// NETWORK 14 (disabled)
//   axisdata[6].Axis_Inbb: A-0-0021.13 -RD- Axis is ready for power to the amplifier (bb)
//   FP_S_0_0095: Diagnostic message
//   drive6: Real axis "Drive6" with axis number 6
// fb_blink_diagnos_6(ENABLE := axisdata[6].Axis_Inbb, TIMELOW := t#1s, TIMEHIGH := t#1s); // BLINK
// fb_diagnose_6(
//     Execute := fb_blink_diagnos_6.OUT,
//     ParameterNumber := FP_S_0_0095,
//     Axis := drive6,
//     Value => str_diagnose_6); // MB_ReadStringParameter

// NETWORK 15
//   axisdata[1].Axis_Inbb: A-0-0021.13 -RD- Axis is ready for power to the amplifier (bb)
//   FP_S_0_0051: Position feedback value 1
//   drive1: Real axis "Drive1" with axis number 1
FB_readmotorencoder1(
    Enable := axisdata[1].Axis_Inbb,
    ParameterNumber := FP_S_0_0051,
    Axis := drive1,
    Value => r_motorencoder_1); // MB_ReadRealParameter

// NETWORK 16
//   axisdata[2].Axis_Inbb: A-0-0021.13 -RD- Axis is ready for power to the amplifier (bb)
//   FP_S_0_0051: Position feedback value 1
//   drive2: Real axis "Drive2" with axis number 2
FB_readmotorencoder2(
    Enable := axisdata[2].Axis_Inbb,
    ParameterNumber := FP_S_0_0051,
    Axis := drive2,
    Value => r_motorencoder_2); // MB_ReadRealParameter

// NETWORK 17
//   axisdata[3].Axis_Inbb: A-0-0021.13 -RD- Axis is ready for power to the amplifier (bb)
//   FP_S_0_0051: Position feedback value 1
//   drive3: Real axis "Drive3" with axis number 3
FB_readmotorencoder3(
    Enable := axisdata[3].Axis_Inbb,
    ParameterNumber := FP_S_0_0051,
    Axis := drive3,
    Value => r_motorencoder_3); // MB_ReadRealParameter

// NETWORK 18 (disabled)
//   axisdata[4].Axis_Inbb: A-0-0021.13 -RD- Axis is ready for power to the amplifier (bb)
//   FP_S_0_0051: Position feedback value 1
//   drive4: Real axis "Drive4" with axis number 4
// FB_readmotorencoder4(
//     Enable := axisdata[4].Axis_Inbb,
//     ParameterNumber := FP_S_0_0051,
//     Axis := drive4,
//     Value => r_motorencoder_4); // MB_ReadRealParameter

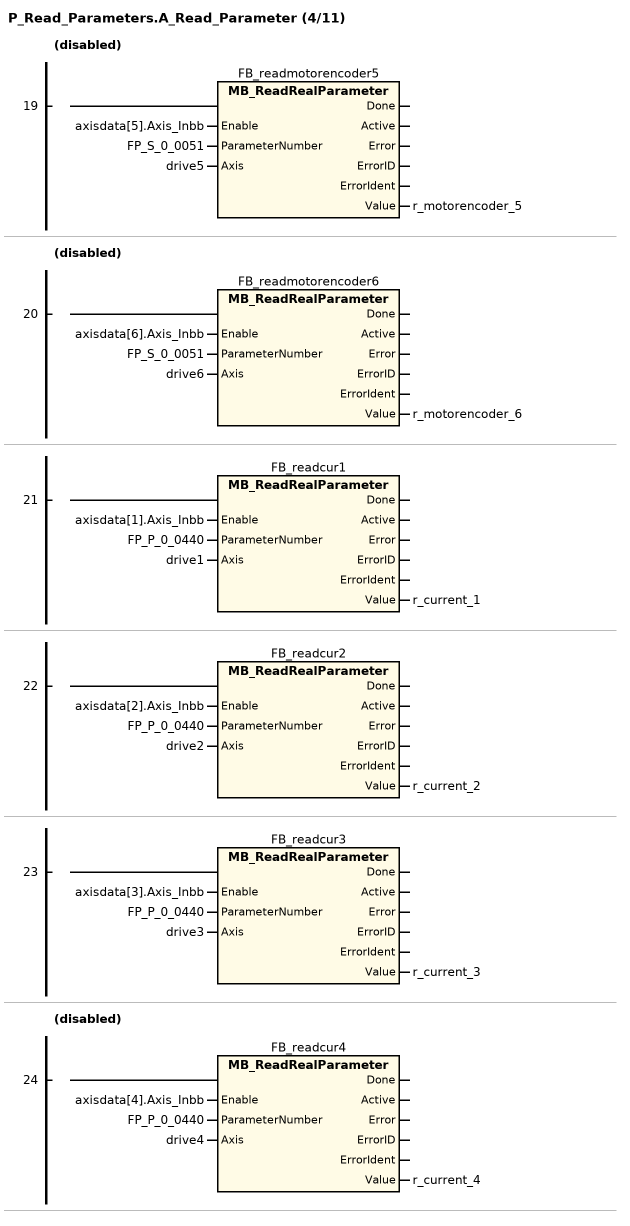
// NETWORK 19 (disabled)
//   axisdata[5].Axis_Inbb: A-0-0021.13 -RD- Axis is ready for power to the amplifier (bb)
//   FP_S_0_0051: Position feedback value 1
//   drive5: Real axis "Drive5" with axis number 5
// FB_readmotorencoder5(
//     Enable := axisdata[5].Axis_Inbb,
//     ParameterNumber := FP_S_0_0051,
//     Axis := drive5,
//     Value => r_motorencoder_5); // MB_ReadRealParameter

// NETWORK 20 (disabled)
//   axisdata[6].Axis_Inbb: A-0-0021.13 -RD- Axis is ready for power to the amplifier (bb)
//   FP_S_0_0051: Position feedback value 1
//   drive6: Real axis "Drive6" with axis number 6
// FB_readmotorencoder6(
//     Enable := axisdata[6].Axis_Inbb,
//     ParameterNumber := FP_S_0_0051,
//     Axis := drive6,
//     Value => r_motorencoder_6); // MB_ReadRealParameter

// NETWORK 21
//   FB_readcur1: With the function block "MB_ReadRealParameter" it is possible to read the current value of a parameter. The return value is REAL.
//   axisdata[1].Axis_Inbb: A-0-0021.13 -RD- Axis is ready for power to the amplifier (bb)
//   FP_P_0_0440: Actual output current value (absolute value)
//   drive1: Real axis "Drive1" with axis number 1
//   r_current_1: FP_P_0_0440,Actual output current value absolute value
FB_readcur1(
    Enable := axisdata[1].Axis_Inbb,
    ParameterNumber := FP_P_0_0440,
    Axis := drive1,
    Value => r_current_1); // MB_ReadRealParameter

// NETWORK 22
//   axisdata[2].Axis_Inbb: A-0-0021.13 -RD- Axis is ready for power to the amplifier (bb)
//   FP_P_0_0440: Actual output current value (absolute value)
//   drive2: Real axis "Drive2" with axis number 2
FB_readcur2(
    Enable := axisdata[2].Axis_Inbb,
    ParameterNumber := FP_P_0_0440,
    Axis := drive2,
    Value => r_current_2); // MB_ReadRealParameter

// NETWORK 23
//   axisdata[3].Axis_Inbb: A-0-0021.13 -RD- Axis is ready for power to the amplifier (bb)
//   FP_P_0_0440: Actual output current value (absolute value)
//   drive3: Real axis "Drive3" with axis number 3
FB_readcur3(
    Enable := axisdata[3].Axis_Inbb,
    ParameterNumber := FP_P_0_0440,
    Axis := drive3,
    Value => r_current_3); // MB_ReadRealParameter

// NETWORK 24 (disabled)
//   axisdata[4].Axis_Inbb: A-0-0021.13 -RD- Axis is ready for power to the amplifier (bb)
//   FP_P_0_0440: Actual output current value (absolute value)
//   drive4: Real axis "Drive4" with axis number 4
// FB_readcur4(
//     Enable := axisdata[4].Axis_Inbb,
//     ParameterNumber := FP_P_0_0440,
//     Axis := drive4,
//     Value => r_current_4); // MB_ReadRealParameter

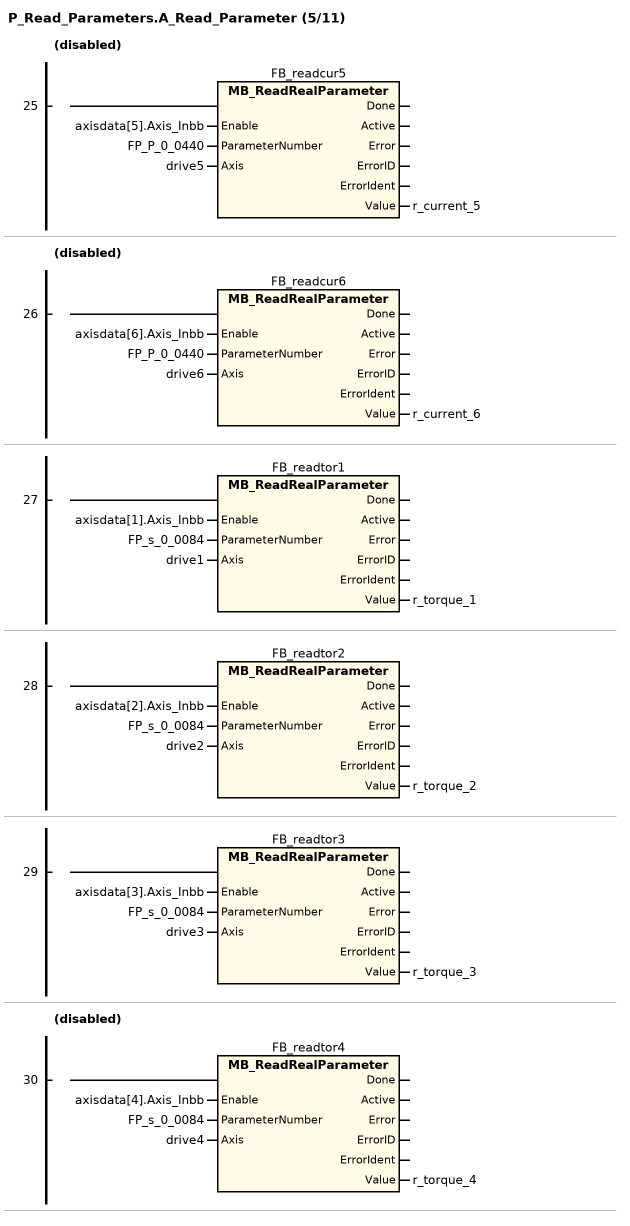
// NETWORK 25 (disabled)
//   axisdata[5].Axis_Inbb: A-0-0021.13 -RD- Axis is ready for power to the amplifier (bb)
//   FP_P_0_0440: Actual output current value (absolute value)
//   drive5: Real axis "Drive5" with axis number 5
// FB_readcur5(
//     Enable := axisdata[5].Axis_Inbb,
//     ParameterNumber := FP_P_0_0440,
//     Axis := drive5,
//     Value => r_current_5); // MB_ReadRealParameter

// NETWORK 26 (disabled)
//   axisdata[6].Axis_Inbb: A-0-0021.13 -RD- Axis is ready for power to the amplifier (bb)
//   FP_P_0_0440: Actual output current value (absolute value)
//   drive6: Real axis "Drive6" with axis number 6
// FB_readcur6(
//     Enable := axisdata[6].Axis_Inbb,
//     ParameterNumber := FP_P_0_0440,
//     Axis := drive6,
//     Value => r_current_6); // MB_ReadRealParameter

// NETWORK 27
//   axisdata[1].Axis_Inbb: A-0-0021.13 -RD- Axis is ready for power to the amplifier (bb)
//   FP_s_0_0084: Torque/force feedback value
//   drive1: Real axis "Drive1" with axis number 1
//   r_torque_1: FP_S_0_0084,Torque force feedback value
FB_readtor1(
    Enable := axisdata[1].Axis_Inbb,
    ParameterNumber := FP_s_0_0084,
    Axis := drive1,
    Value => r_torque_1); // MB_ReadRealParameter

// NETWORK 28
//   axisdata[2].Axis_Inbb: A-0-0021.13 -RD- Axis is ready for power to the amplifier (bb)
//   FP_s_0_0084: Torque/force feedback value
//   drive2: Real axis "Drive2" with axis number 2
FB_readtor2(
    Enable := axisdata[2].Axis_Inbb,
    ParameterNumber := FP_s_0_0084,
    Axis := drive2,
    Value => r_torque_2); // MB_ReadRealParameter

// NETWORK 29
//   axisdata[3].Axis_Inbb: A-0-0021.13 -RD- Axis is ready for power to the amplifier (bb)
//   FP_s_0_0084: Torque/force feedback value
//   drive3: Real axis "Drive3" with axis number 3
FB_readtor3(
    Enable := axisdata[3].Axis_Inbb,
    ParameterNumber := FP_s_0_0084,
    Axis := drive3,
    Value => r_torque_3); // MB_ReadRealParameter

// NETWORK 30 (disabled)
//   axisdata[4].Axis_Inbb: A-0-0021.13 -RD- Axis is ready for power to the amplifier (bb)
//   FP_s_0_0084: Torque/force feedback value
//   drive4: Real axis "Drive4" with axis number 4
// FB_readtor4(
//     Enable := axisdata[4].Axis_Inbb,
//     ParameterNumber := FP_s_0_0084,
//     Axis := drive4,
//     Value => r_torque_4); // MB_ReadRealParameter

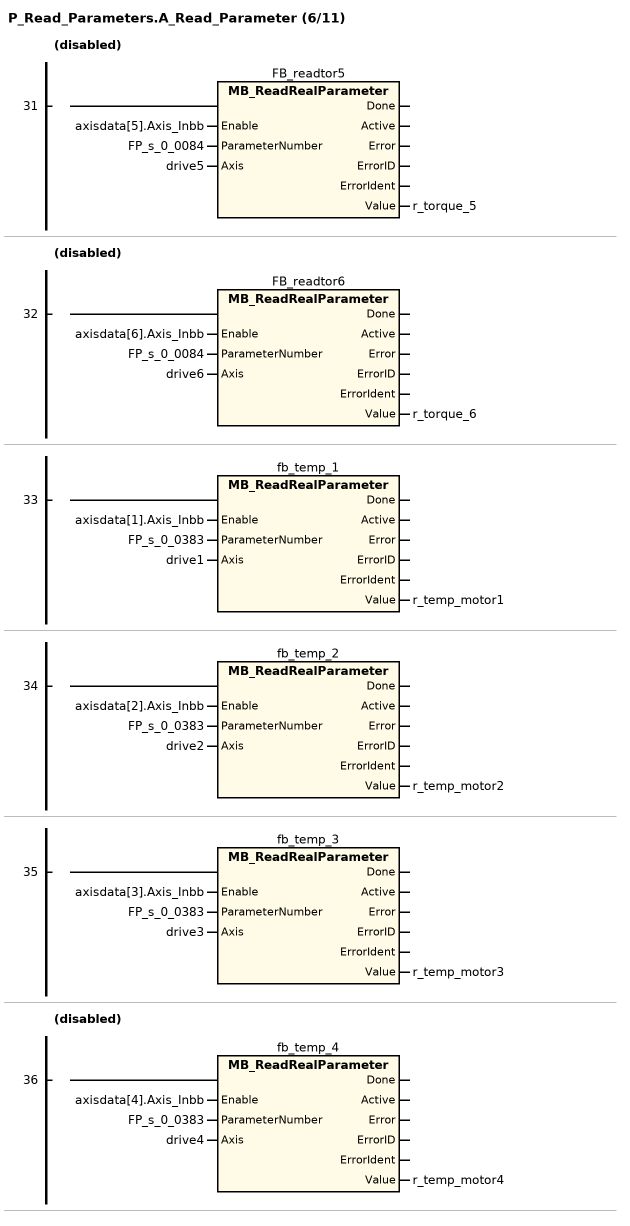
// NETWORK 31 (disabled)
//   axisdata[5].Axis_Inbb: A-0-0021.13 -RD- Axis is ready for power to the amplifier (bb)
//   FP_s_0_0084: Torque/force feedback value
//   drive5: Real axis "Drive5" with axis number 5
// FB_readtor5(
//     Enable := axisdata[5].Axis_Inbb,
//     ParameterNumber := FP_s_0_0084,
//     Axis := drive5,
//     Value => r_torque_5); // MB_ReadRealParameter

// NETWORK 32 (disabled)
//   axisdata[6].Axis_Inbb: A-0-0021.13 -RD- Axis is ready for power to the amplifier (bb)
//   FP_s_0_0084: Torque/force feedback value
//   drive6: Real axis "Drive6" with axis number 6
// FB_readtor6(
//     Enable := axisdata[6].Axis_Inbb,
//     ParameterNumber := FP_s_0_0084,
//     Axis := drive6,
//     Value => r_torque_6); // MB_ReadRealParameter

// NETWORK 33
//   axisdata[1].Axis_Inbb: A-0-0021.13 -RD- Axis is ready for power to the amplifier (bb)
//   FP_s_0_0383: Motor temperature
//   drive1: Real axis "Drive1" with axis number 1
//   r_temp_motor1: FP_S_0_0383,Motor temperature
fb_temp_1(
    Enable := axisdata[1].Axis_Inbb,
    ParameterNumber := FP_s_0_0383,
    Axis := drive1,
    Value => r_temp_motor1); // MB_ReadRealParameter

// NETWORK 34
//   axisdata[2].Axis_Inbb: A-0-0021.13 -RD- Axis is ready for power to the amplifier (bb)
//   FP_s_0_0383: Motor temperature
//   drive2: Real axis "Drive2" with axis number 2
fb_temp_2(
    Enable := axisdata[2].Axis_Inbb,
    ParameterNumber := FP_s_0_0383,
    Axis := drive2,
    Value => r_temp_motor2); // MB_ReadRealParameter

// NETWORK 35
//   axisdata[3].Axis_Inbb: A-0-0021.13 -RD- Axis is ready for power to the amplifier (bb)
//   FP_s_0_0383: Motor temperature
//   drive3: Real axis "Drive3" with axis number 3
fb_temp_3(
    Enable := axisdata[3].Axis_Inbb,
    ParameterNumber := FP_s_0_0383,
    Axis := drive3,
    Value => r_temp_motor3); // MB_ReadRealParameter

// NETWORK 36 (disabled)
//   axisdata[4].Axis_Inbb: A-0-0021.13 -RD- Axis is ready for power to the amplifier (bb)
//   FP_s_0_0383: Motor temperature
//   drive4: Real axis "Drive4" with axis number 4
// fb_temp_4(
//     Enable := axisdata[4].Axis_Inbb,
//     ParameterNumber := FP_s_0_0383,
//     Axis := drive4,
//     Value => r_temp_motor4); // MB_ReadRealParameter

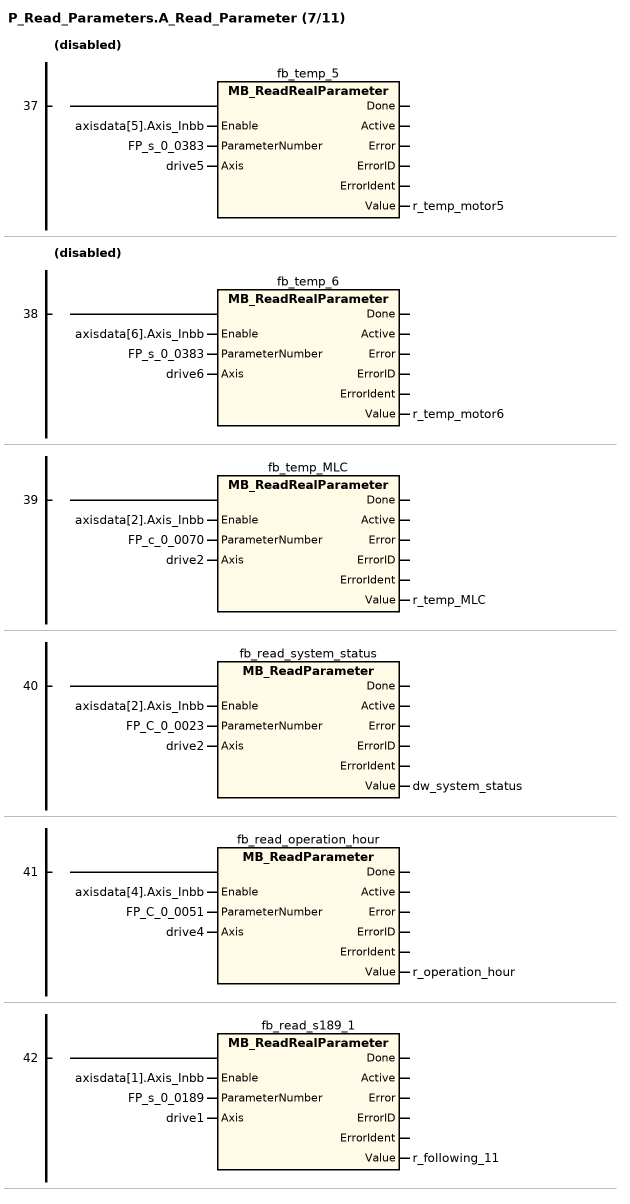
// NETWORK 37 (disabled)
//   axisdata[5].Axis_Inbb: A-0-0021.13 -RD- Axis is ready for power to the amplifier (bb)
//   FP_s_0_0383: Motor temperature
//   drive5: Real axis "Drive5" with axis number 5
// fb_temp_5(
//     Enable := axisdata[5].Axis_Inbb,
//     ParameterNumber := FP_s_0_0383,
//     Axis := drive5,
//     Value => r_temp_motor5); // MB_ReadRealParameter

// NETWORK 38 (disabled)
//   axisdata[6].Axis_Inbb: A-0-0021.13 -RD- Axis is ready for power to the amplifier (bb)
//   FP_s_0_0383: Motor temperature
//   drive6: Real axis "Drive6" with axis number 6
// fb_temp_6(
//     Enable := axisdata[6].Axis_Inbb,
//     ParameterNumber := FP_s_0_0383,
//     Axis := drive6,
//     Value => r_temp_motor6); // MB_ReadRealParameter

// NETWORK 39
//   fb_temp_MLC: <<<<<<<<<<<<<<<<<<<<<<<<<<<<<<<<<<<<<<<add MLC temperature and operation hour(20100708)>>>>>>>>>>>>>>>>>>>>>>>>>>>>>>>>>>>>>
//   axisdata[2].Axis_Inbb: A-0-0021.13 -RD- Axis is ready for power to the amplifier (bb)
//   FP_c_0_0070: Control temperature
//   drive2: Real axis "Drive2" with axis number 2
//   r_temp_MLC: FP_c_0_0070,Control unit temperature
fb_temp_MLC(
    Enable := axisdata[2].Axis_Inbb,
    ParameterNumber := FP_c_0_0070,
    Axis := drive2,
    Value => r_temp_MLC); // MB_ReadRealParameter

// NETWORK 40
//   axisdata[2].Axis_Inbb: A-0-0021.13 -RD- Axis is ready for power to the amplifier (bb)
//   FP_C_0_0023: System status
//   drive2: Real axis "Drive2" with axis number 2
//   dw_system_status: FP_C_0_0023,MC system status,used for temperature warning
fb_read_system_status(
    Enable := axisdata[2].Axis_Inbb,
    ParameterNumber := FP_C_0_0023,
    Axis := drive2,
    Value => dw_system_status); // MB_ReadParameter

// NETWORK 41
//   axisdata[4].Axis_Inbb: A-0-0021.13 -RD- Axis is ready for power to the amplifier (bb)
//   FP_C_0_0051: Operating hour counter
//   drive4: Real axis "Drive4" with axis number 4
//   r_operation_hour: FP_C_0_0051,Operation hour counter
fb_read_operation_hour(
    Enable := axisdata[4].Axis_Inbb,
    ParameterNumber := FP_C_0_0051,
    Axis := drive4,
    Value => r_operation_hour); // MB_ReadParameter

// NETWORK 42
//   axisdata[1].Axis_Inbb: A-0-0021.13 -RD- Axis is ready for power to the amplifier (bb)
//   FP_s_0_0189: Following distance
//   drive1: Real axis "Drive1" with axis number 1
//   r_following_11: FP_s_0_0189,following error
fb_read_s189_1(
    Enable := axisdata[1].Axis_Inbb,
    ParameterNumber := FP_s_0_0189,
    Axis := drive1,
    Value => r_following_11); // MB_ReadRealParameter

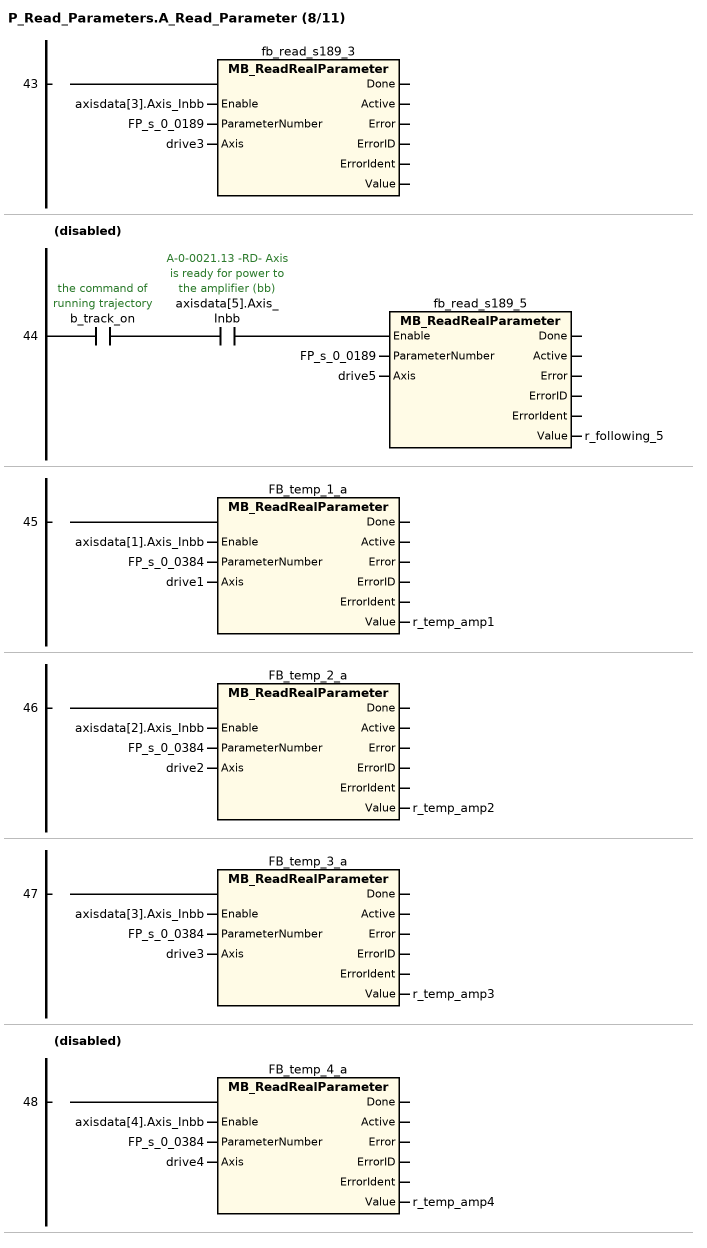
// NETWORK 43
//   axisdata[3].Axis_Inbb: A-0-0021.13 -RD- Axis is ready for power to the amplifier (bb)
//   FP_s_0_0189: Following distance
//   drive3: Real axis "Drive3" with axis number 3
fb_read_s189_3(Enable := axisdata[3].Axis_Inbb, ParameterNumber := FP_s_0_0189, Axis := drive3); // MB_ReadRealParameter

// NETWORK 44 (disabled)
//   b_track_on: the command of running trajectory
//   axisdata[5].Axis_Inbb: A-0-0021.13 -RD- Axis is ready for power to the amplifier (bb)
//   FP_s_0_0189: Following distance
//   drive5: Real axis "Drive5" with axis number 5
// fb_read_s189_5(
//     Enable := b_track_on AND axisdata[5].Axis_Inbb,
//     ParameterNumber := FP_s_0_0189,
//     Axis := drive5,
//     Value => r_following_5); // MB_ReadRealParameter

// NETWORK 45
//   axisdata[1].Axis_Inbb: A-0-0021.13 -RD- Axis is ready for power to the amplifier (bb)
//   FP_s_0_0384: Amplifier temperature
//   drive1: Real axis "Drive1" with axis number 1
//   r_temp_amp1: FP_S_0_0384,Amplifier temperature
FB_temp_1_a(
    Enable := axisdata[1].Axis_Inbb,
    ParameterNumber := FP_s_0_0384,
    Axis := drive1,
    Value => r_temp_amp1); // MB_ReadRealParameter

// NETWORK 46
//   axisdata[2].Axis_Inbb: A-0-0021.13 -RD- Axis is ready for power to the amplifier (bb)
//   FP_s_0_0384: Amplifier temperature
//   drive2: Real axis "Drive2" with axis number 2
FB_temp_2_a(
    Enable := axisdata[2].Axis_Inbb,
    ParameterNumber := FP_s_0_0384,
    Axis := drive2,
    Value => r_temp_amp2); // MB_ReadRealParameter

// NETWORK 47
//   axisdata[3].Axis_Inbb: A-0-0021.13 -RD- Axis is ready for power to the amplifier (bb)
//   FP_s_0_0384: Amplifier temperature
//   drive3: Real axis "Drive3" with axis number 3
FB_temp_3_a(
    Enable := axisdata[3].Axis_Inbb,
    ParameterNumber := FP_s_0_0384,
    Axis := drive3,
    Value => r_temp_amp3); // MB_ReadRealParameter

// NETWORK 48 (disabled)
//   axisdata[4].Axis_Inbb: A-0-0021.13 -RD- Axis is ready for power to the amplifier (bb)
//   FP_s_0_0384: Amplifier temperature
//   drive4: Real axis "Drive4" with axis number 4
// FB_temp_4_a(
//     Enable := axisdata[4].Axis_Inbb,
//     ParameterNumber := FP_s_0_0384,
//     Axis := drive4,
//     Value => r_temp_amp4); // MB_ReadRealParameter

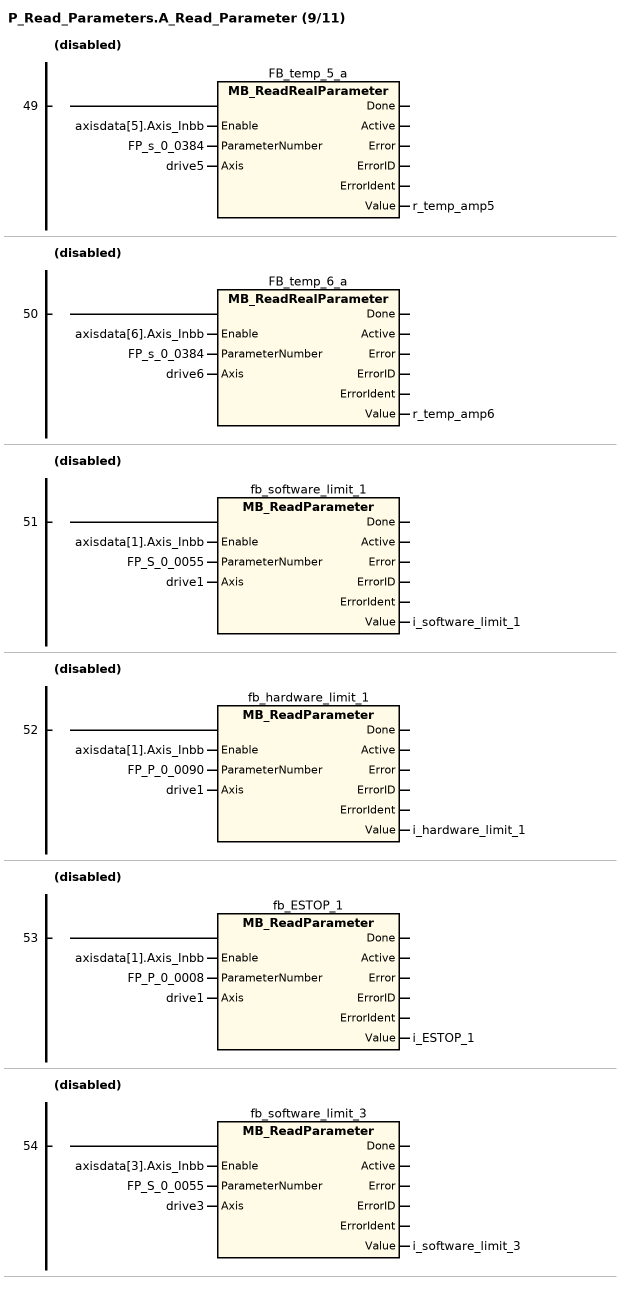
// NETWORK 49 (disabled)
//   axisdata[5].Axis_Inbb: A-0-0021.13 -RD- Axis is ready for power to the amplifier (bb)
//   FP_s_0_0384: Amplifier temperature
//   drive5: Real axis "Drive5" with axis number 5
// FB_temp_5_a(
//     Enable := axisdata[5].Axis_Inbb,
//     ParameterNumber := FP_s_0_0384,
//     Axis := drive5,
//     Value => r_temp_amp5); // MB_ReadRealParameter

// NETWORK 50 (disabled)
//   axisdata[6].Axis_Inbb: A-0-0021.13 -RD- Axis is ready for power to the amplifier (bb)
//   FP_s_0_0384: Amplifier temperature
//   drive6: Real axis "Drive6" with axis number 6
// FB_temp_6_a(
//     Enable := axisdata[6].Axis_Inbb,
//     ParameterNumber := FP_s_0_0384,
//     Axis := drive6,
//     Value => r_temp_amp6); // MB_ReadRealParameter

// NETWORK 51 (disabled)
//   fb_software_limit_1: test for limit check
//   axisdata[1].Axis_Inbb: A-0-0021.13 -RD- Axis is ready for power to the amplifier (bb)
//   FP_S_0_0055: Position polarities
//   drive1: Real axis "Drive1" with axis number 1
// fb_software_limit_1(
//     Enable := axisdata[1].Axis_Inbb,
//     ParameterNumber := FP_S_0_0055,
//     Axis := drive1,
//     Value => i_software_limit_1); // MB_ReadParameter

// NETWORK 52 (disabled)
//   axisdata[1].Axis_Inbb: A-0-0021.13 -RD- Axis is ready for power to the amplifier (bb)
//   FP_P_0_0090: Travel range limit parameter
//   drive1: Real axis "Drive1" with axis number 1
// fb_hardware_limit_1(
//     Enable := axisdata[1].Axis_Inbb,
//     ParameterNumber := FP_P_0_0090,
//     Axis := drive1,
//     Value => i_hardware_limit_1); // MB_ReadParameter

// NETWORK 53 (disabled)
//   axisdata[1].Axis_Inbb: A-0-0021.13 -RD- Axis is ready for power to the amplifier (bb)
//   FP_P_0_0008: Activation E-Stop function
//   drive1: Real axis "Drive1" with axis number 1
// fb_ESTOP_1(
//     Enable := axisdata[1].Axis_Inbb,
//     ParameterNumber := FP_P_0_0008,
//     Axis := drive1,
//     Value => i_ESTOP_1); // MB_ReadParameter

// NETWORK 54 (disabled)
//   axisdata[3].Axis_Inbb: A-0-0021.13 -RD- Axis is ready for power to the amplifier (bb)
//   FP_S_0_0055: Position polarities
//   drive3: Real axis "Drive3" with axis number 3
// fb_software_limit_3(
//     Enable := axisdata[3].Axis_Inbb,
//     ParameterNumber := FP_S_0_0055,
//     Axis := drive3,
//     Value => i_software_limit_3); // MB_ReadParameter

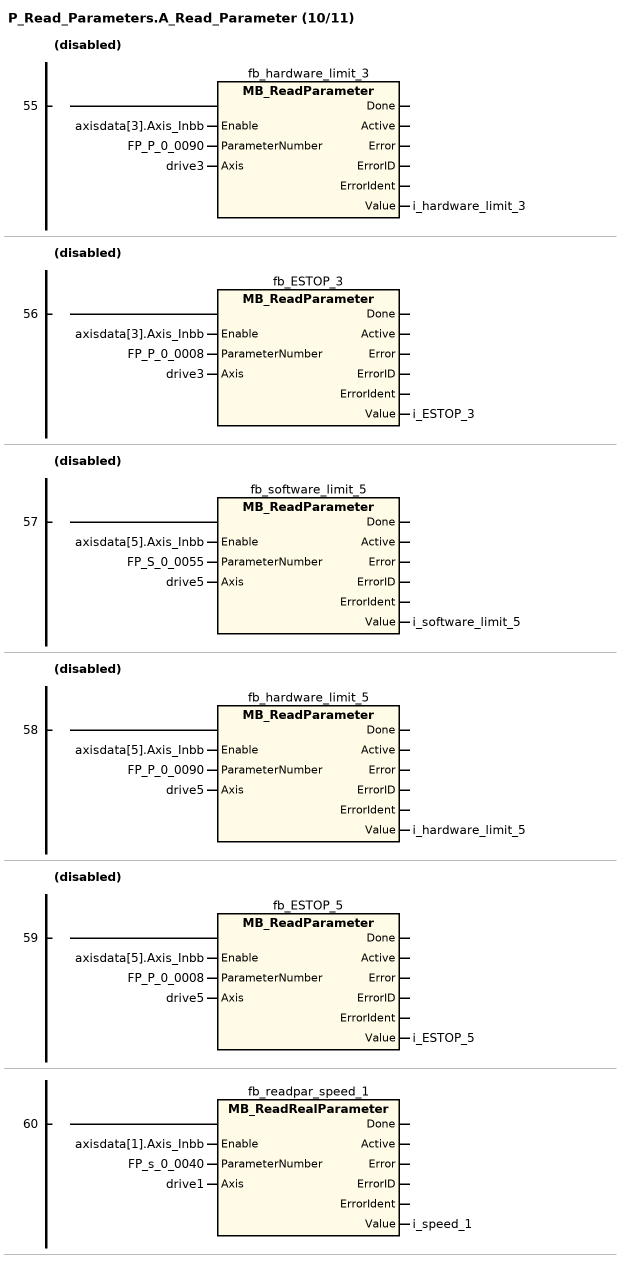
// NETWORK 55 (disabled)
//   axisdata[3].Axis_Inbb: A-0-0021.13 -RD- Axis is ready for power to the amplifier (bb)
//   FP_P_0_0090: Travel range limit parameter
//   drive3: Real axis "Drive3" with axis number 3
// fb_hardware_limit_3(
//     Enable := axisdata[3].Axis_Inbb,
//     ParameterNumber := FP_P_0_0090,
//     Axis := drive3,
//     Value => i_hardware_limit_3); // MB_ReadParameter

// NETWORK 56 (disabled)
//   axisdata[3].Axis_Inbb: A-0-0021.13 -RD- Axis is ready for power to the amplifier (bb)
//   FP_P_0_0008: Activation E-Stop function
//   drive3: Real axis "Drive3" with axis number 3
// fb_ESTOP_3(
//     Enable := axisdata[3].Axis_Inbb,
//     ParameterNumber := FP_P_0_0008,
//     Axis := drive3,
//     Value => i_ESTOP_3); // MB_ReadParameter

// NETWORK 57 (disabled)
//   axisdata[5].Axis_Inbb: A-0-0021.13 -RD- Axis is ready for power to the amplifier (bb)
//   FP_S_0_0055: Position polarities
//   drive5: Real axis "Drive5" with axis number 5
// fb_software_limit_5(
//     Enable := axisdata[5].Axis_Inbb,
//     ParameterNumber := FP_S_0_0055,
//     Axis := drive5,
//     Value => i_software_limit_5); // MB_ReadParameter

// NETWORK 58 (disabled)
//   axisdata[5].Axis_Inbb: A-0-0021.13 -RD- Axis is ready for power to the amplifier (bb)
//   FP_P_0_0090: Travel range limit parameter
//   drive5: Real axis "Drive5" with axis number 5
// fb_hardware_limit_5(
//     Enable := axisdata[5].Axis_Inbb,
//     ParameterNumber := FP_P_0_0090,
//     Axis := drive5,
//     Value => i_hardware_limit_5); // MB_ReadParameter

// NETWORK 59 (disabled)
//   axisdata[5].Axis_Inbb: A-0-0021.13 -RD- Axis is ready for power to the amplifier (bb)
//   FP_P_0_0008: Activation E-Stop function
//   drive5: Real axis "Drive5" with axis number 5
// fb_ESTOP_5(
//     Enable := axisdata[5].Axis_Inbb,
//     ParameterNumber := FP_P_0_0008,
//     Axis := drive5,
//     Value => i_ESTOP_5); // MB_ReadParameter

// NETWORK 60
//   axisdata[1].Axis_Inbb: A-0-0021.13 -RD- Axis is ready for power to the amplifier (bb)
//   FP_s_0_0040: Velocity feedback value
//   drive1: Real axis "Drive1" with axis number 1
//   i_speed_1: the velocity feedback value of motor1
fb_readpar_speed_1(
    Enable := axisdata[1].Axis_Inbb,
    ParameterNumber := FP_s_0_0040,
    Axis := drive1,
    Value => i_speed_1); // MB_ReadRealParameter

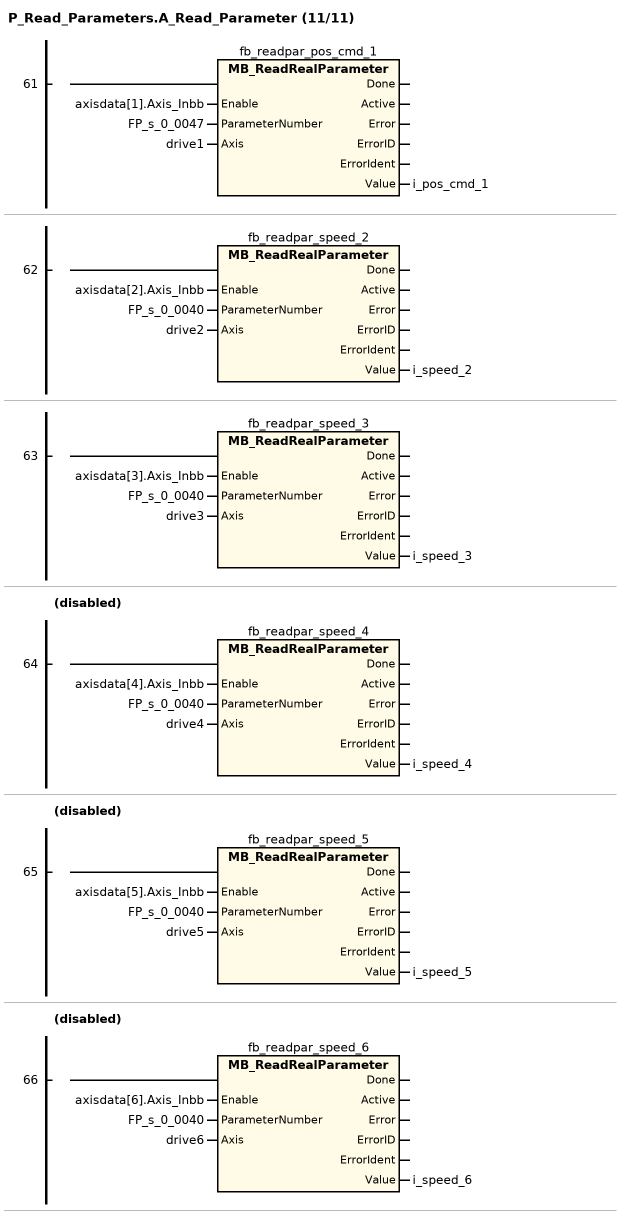
// NETWORK 61
//   axisdata[1].Axis_Inbb: A-0-0021.13 -RD- Axis is ready for power to the amplifier (bb)
//   FP_s_0_0047: Velocity feedback value
//   drive1: Real axis "Drive1" with axis number 1
//   i_pos_cmd_1: the velocity feedback value of motor1
fb_readpar_pos_cmd_1(
    Enable := axisdata[1].Axis_Inbb,
    ParameterNumber := FP_s_0_0047,
    Axis := drive1,
    Value => i_pos_cmd_1); // MB_ReadRealParameter

// NETWORK 62
//   axisdata[2].Axis_Inbb: A-0-0021.13 -RD- Axis is ready for power to the amplifier (bb)
//   FP_s_0_0040: Velocity feedback value
//   drive2: Real axis "Drive2" with axis number 2
//   i_speed_2: the velocity feedback value of motor1
fb_readpar_speed_2(
    Enable := axisdata[2].Axis_Inbb,
    ParameterNumber := FP_s_0_0040,
    Axis := drive2,
    Value => i_speed_2); // MB_ReadRealParameter

// NETWORK 63
//   axisdata[3].Axis_Inbb: A-0-0021.13 -RD- Axis is ready for power to the amplifier (bb)
//   FP_s_0_0040: Velocity feedback value
//   drive3: Real axis "Drive3" with axis number 3
//   i_speed_3: the velocity feedback value of motor3
fb_readpar_speed_3(
    Enable := axisdata[3].Axis_Inbb,
    ParameterNumber := FP_s_0_0040,
    Axis := drive3,
    Value => i_speed_3); // MB_ReadRealParameter

// NETWORK 64 (disabled)
//   axisdata[4].Axis_Inbb: A-0-0021.13 -RD- Axis is ready for power to the amplifier (bb)
//   FP_s_0_0040: Velocity feedback value
//   drive4: Real axis "Drive4" with axis number 4
//   i_speed_4: the velocity feedback value of motor1
// fb_readpar_speed_4(
//     Enable := axisdata[4].Axis_Inbb,
//     ParameterNumber := FP_s_0_0040,
//     Axis := drive4,
//     Value => i_speed_4); // MB_ReadRealParameter

// NETWORK 65 (disabled)
//   axisdata[5].Axis_Inbb: A-0-0021.13 -RD- Axis is ready for power to the amplifier (bb)
//   FP_s_0_0040: Velocity feedback value
//   drive5: Real axis "Drive5" with axis number 5
//   i_speed_5: the velocity feedback value of motor5
// fb_readpar_speed_5(
//     Enable := axisdata[5].Axis_Inbb,
//     ParameterNumber := FP_s_0_0040,
//     Axis := drive5,
//     Value => i_speed_5); // MB_ReadRealParameter

// NETWORK 66 (disabled)
//   axisdata[6].Axis_Inbb: A-0-0021.13 -RD- Axis is ready for power to the amplifier (bb)
//   FP_s_0_0040: Velocity feedback value
//   drive6: Real axis "Drive6" with axis number 6
//   i_speed_6: the velocity feedback value of motor1
// fb_readpar_speed_6(
//     Enable := axisdata[6].Axis_Inbb,
//     ParameterNumber := FP_s_0_0040,
//     Axis := drive6,
//     Value => i_speed_6); // MB_ReadRealParameter
END_ACTION

END_PROGRAM

// IndraMotionMlc1/Application/POUs/Motion/P_interpolator
(*This program is built for running trajectory,and the trajectory runs by the rule y=ax^2+bx+c.
In this PROGRAM,there are two kinds OF FUNCTION blocks,ML_WriteCyclicPosition AND ML_OpenCyclicPositionChannel.
They are used for give the position command value to the virtual axis.*)
PROGRAM P_interpolator
VAR
(*azimuth,elevation and FeedIndexer position at i_start point *)
	p1_az: LREAL;
	p1_el: LREAL;
	p1_FI: LREAL;
(*azimuth,elevation and FeedIndexer position at i_start+1 point*)
	p2_az: LREAL;
	p2_el: LREAL;
	p2_FI: LREAL;
(*azimuth,elevation and FeedIndexer position at i_start+2 point*)
	p3_az: LREAL;
	p3_el: LREAL;
	p3_FI: LREAL;
(*the facters of the formula y=ax^2+bx+c*)
	a_az: LREAL;
	b_az: LREAL;
	a_el: LREAL;
	b_el: LREAL;
	a_FI: LREAL;
	b_FI: LREAL;
	t: LREAL;
	t1: LREAL;(*the time at i_start point*)
	t2: LREAL;(*the time at i_start+1 point*)
	t3: LREAL;(*the time at i_start+2 point*)
	
(*<<<<<<<<<<<<<<<<<<<<<<<<Write a Position value to azimuth,elevation and FeedIndexer virtual axis>>>>>>>>>>>>>>>>>>*)
	fb_write_positon_az: ML_WriteCyclicPosition;
	fb_write_positon_el: ML_WriteCyclicPosition;
	fb_write_positon_FI: ML_WriteCyclicPosition;

(*Open Cyclic Position Channel for azimuth,elevation and FeedIndexer.
Only if the cyclic position target value channel is open, 
the position command will become effective in the next cycle on the axis.*)
	fb_open_channel_az: ML_OpenCyclicPositionChannel;
	fb_open_channel_el: ML_OpenCyclicPositionChannel;
	fb_open_channel_FI: ML_OpenCyclicPositionChannel;

(*<<<<<<<<<<<<<definition for rtrig>>>>>>>>>>>>>>*)
	rtrig_track_on: R_TRIG;
	rtrig_write_position: R_TRIG;
	rtrig_reset_open_channel: R_TRIG;
	rtrig_reset_goto_track: R_TRIG;
	r_rtrig_start_stop:R_TRIG;
	ton_track_on:TON;
	b_signal_for_open: BOOL;
(*<<<<<<<<<<<<<<<<<<<<<<<the current position>>>>>>>>>>>>>>>>>>>*)
	r_last_position_az: LREAL;
	r_last_position_el: LREAL;
	r_last_position_FI: LREAL;
(*<<<<<<<<<<<<<<<<<<<<<<<<<<the current speed>>>>>>>>>>>>>>>>>>>>*)
	r_vel_last_az: LREAL;
	r_vel_last_el: LREAL;
	r_vel_last_FI: LREAL;
(*the distance and time between the current point and the first point*)
	r_start_distance_az: LREAL;
	r_start_distance_el: LREAL;
	r_start_distance_FI: LREAL;
	r_time_distance: LREAL;
(*the current velocity *)
	r_vel_start_az: LREAL;
	r_vel_start_el: LREAL;
	r_vel_start_FI: LREAL;
(*the transition for the azimuth position,r_write_position_az.*)
	r_calc_pos_az:LREAL;
	V0_el: LREAL;
	V0_az: LREAL;
	V0_FI: LREAL;
	i_point_caught: INT:=1;
	V_start_az: LREAL;
	V_start_el: LREAL;
	V_start_FI: LREAL;
	i_caught_MJD1:LREAL;
	i_caught_MJD2:LREAL;
	i_caught_TAIoffset1:LREAL;
	i_caught_TAIoffset2:LREAL;
	b_test:BOOL;
	
	i_start_first:INT;
	i_end_first:INT;
	
	test_1:INT;
	test_2:INT;
	
	r_start_az:LREAL;
	r_caught_az:LREAL;
	
	ton_pause_on:TON;
	rtrig_pause_on:R_TRIG;
	r_abs_az_speed:LREAL; // units deg/sec
	r_abs_el_speed:LREAL; // units deg/sec
	test_enable_el: BOOL;
	b_start_to_compensate: BOOL;
	p_covert_velocity:LREAL;
	r_following_test: LREAL;
	r_following_31: LREAL;
	r_following_333: LREAL;
	p_covert_velocity_el: LREAL;	
	(**********offset************)
	r_az_offset_Vmax:LREAL:=2.0;
	r_el_offset_Vmax:LREAL:=0.85;
	r_az_offset_acc:LREAL:=1.0;
	r_el_offset_acc:LREAL:=0.25;
	r_az_offset_dec:LREAL:=0.5;
	r_el_offset_dec:LREAL:=0.25;
	r_old_offset_az:LREAL;
	r_old_offset_el:LREAL;
	r_new_offset_az:LREAL;
	r_new_offset_el:LREAL;

	r_test_offset_az_abs:LREAL;
	r_test_offset_el_abs:LREAL;
	i_test_offset_count:DINT:=0;
	r_offset_t1_acc:LREAL;
	r_offset_t2_v:LREAL;
	r_offset_t3_dec:LREAL;
	l_offset_t1_acc:LREAL;
	l_offset_t2_v:LREAL;
	l_offset_t3_dec:LREAL;
	r_offset_t1_acc_el:LREAL;
	r_offset_t2_v_el:LREAL;
	r_offset_t3_dec_el:LREAL;
	l_offset_t1_acc_el:LREAL;
	l_offset_t2_v_el:LREAL;
	l_offset_t3_dec_el:LREAL;
	r_offset_t:LREAL:=0;
	test_t:LREAL;
	r_az_offset_abs:LREAL;
	
	Static_done: BOOL;
	r_write_position_az_s: LREAL;
	r_write_position_el_s: LREAL;
	s_mp: StaticPmParam;
	Az_rad: LREAL;
	El_rad: LREAL;
	ABphi_rad: LREAL;
	TE: INT;
	//r_write_position_az_out: LREAL;
	//r_write_position_el_out: LREAL;
	test1: BOOL;
	Test2: BOOL;
	test3: BOOL;
	test4: BOOL;
	test5: BOOL;
	test6: BOOL;
	test7: BOOL;
	test8: BOOL;
	test9: BOOL;
	rtrig_write_position_sim: R_TRIG;
	fb_move_sim_track_Az: MC_MoveAbsolute;
	b_sim_trk_az_done: BOOL;
	b_sim_trk_el_done: BOOL;
	rtrig_reset_sim: R_TRIG;
	rtrig_reset_sim_move: R_TRIG;
	fb_move_sim_track_El: MC_MoveAbsolute;
	b_sim_write_az: BOOL;
	b_sim_trk_az_active: BOOL;
	TON_0: TON;
	b_sim_trk_el_active: BOOL;
	b_sim_trk_az_active_not: BOOL;
	f_trig_sim: F_TRIG;
	R_TRIG_0: R_TRIG;
	F_TRIG_0: F_TRIG;
	F_TRIG_1: F_TRIG;
	TON_1: TON;
	IL_EnableInOpBase_0: IL_SIGNALGENERATORTYPE01;
	TP_0: TP;
	TP_1: TP;
	TP_2: TP;
	BLINK_0: BLINK;
	b_sim_trk_exec: BOOL;
END_VAR

(*IF test_enable_el THEN
arAxisCtrl_gb[Drive3.AxisNo].Admin._OpMode.en := Modeah;
ELSE
arAxisCtrl_gb[Drive3.AxisNo].Admin._OpMode.en := Modeab;
END_IF
*)
//axisdata[3].dwUserCmdDataA_q.REAL_;

//axisdata[3].dwUserActualDataA_i.REAL_;



//axisdata[3].dwUserCmdDataA_q.REAL_:=axisdata[3].dwUserActualDataA_i.REAL_;





(*<<<<<<<<<<<<<<<<<<<<<calculate the current point in the stack>>>>>>>>>>>>>>>>>>>>>>>*)
//WHILE lr_MJD_current >= track_table[F_I_number(i_start+1)].MJD DO
test1:=lr_TAIoffset_current >= track_table[F_I_number(i_start+1)].TAIoffset;
WHILE lr_TAIoffset_current >= track_table[F_I_number(i_start+1)].TAIoffset DO
	IF i_start= i_end THEN
		EXIT;
	ELSE
		i_start:=F_I_number(i_start+1);
	END_IF;
END_WHILE


(*<<<<<<<<<<<<<<<<<<calculate the number of the points left in the stack>>>>>>>>>>>>>>*)
IF i_start=i_end THEN
	i_num_stack_left:=0;
ELSE
	i_num_stack_left:= i_end-i_start+1;
	IF i_num_stack_left<=0 THEN
		i_num_stack_left:=i_num_stack_left+i_total;
	END_IF;
END_IF

(* I Don't know what this piece of code is meant to do commenting it out 8/8/2024
IF i_num_stack_left>10 AND b_remote_on_run AND b_track_on=FALSE THEN
	b_track_on:=TRUE;
END_IF; *)


r_abs_az_speed:=ABS(AxisData[1].rActualVelocity_i)*6;
p_covert_velocity:=(0.5773*r_abs_az_speed*r_abs_az_speed*r_abs_az_speed - 0.4526*r_abs_az_speed*r_abs_az_speed + 11.313*r_abs_az_speed + 4.523)*0.2535;
p_covert_velocity_el:=0.5773*r_vel_EL*r_vel_EL*r_vel_EL - 0.4526*r_vel_EL*r_vel_EL + 11.313*r_vel_EL + 4.523;
(*<<<<<<<<<<<<<<<<<<<<<<<<<<<<<<<<<<<<<<the definication of trigger and TON>>>>>>>>>>>>>>>>>>>>>>>>>>>>>>>>>>>>>>>>>>>>>>>*)
r_rtrig_start_stop(clk:=b_track_on);(*before tracking ,stop the motion*)
ton_track_on(IN:=b_track_on,PT:=T#200MS);(*by using 200ms,program can search about 60 points*)
rtrig_track_on(clk:=ton_track_on.Q);(*the trigger for the initializtion*)


ton_pause_on(IN:=b_Track_Pause,PT:=T#4000MS);(*by using 200ms,program can search about 60 points*)
rtrig_pause_on(clk:=ton_pause_on.Q);(*the trigger for the initializtion*)

IF rtrig_pause_on.Q THEN
	b_track_on:=FALSE;
END_IF


(*<<<<<<<<<<<<<<<<<<<<<<<<<<<<main program of track>>>>>>>>>>>>>>>>>>>>>>>>>>>>>*)
IF b_track_on=TRUE THEN
	
(*<<<<<<<<<<<<<<<<<<<<<<<<<<< Calculate the tracking error>>>>>>>>>>>>>>>>>>>>>>>>>>>>>*)
	
	//IF ABS(track_table[i_start].MJD-lr_mjd_current)*86400<0.001 THEN
	Test2:=ABS(track_table[i_start].TAIoffset-lr_TAIoffset_current)<0.001;
	IF ABS(track_table[i_start].TAIoffset-lr_TAIoffset_current)<0.001 THEN
		r_following_1:=(r_pos_az_v-track_table[i_start].Azimuth);
		IF  ABS(r_following_1)<0.5  THEN
		   r_following_1:=(r_pos_az_v-track_table[i_start].Azimuth)/p_covert_velocity;
		END_IF
		   r_following_3:=(r_pos_el_v-track_table[i_start].Elevation);
		IF ABS(r_following_3)>0.0001 AND ABS(r_following_3)<=0.003 THEN
			r_following_3:=(r_pos_el_v-track_table[i_start].Elevation)/1.5;
		END_IF
		IF ABS(r_following_3)>0.003 AND ABS(r_following_3)<=0.006 THEN
			r_following_3:=(r_pos_el_v-track_table[i_start].Elevation)/2;
		END_IF
		IF ABS(r_following_3)>0.006 AND ABS(r_following_3)<=0.02 THEN
			r_following_3:=(r_pos_el_v-track_table[i_start].Elevation)/4;
		END_IF
		r_following_radius_asec := LREAL_TO_REAL((SQRT(EXPT(r_following_1,2)+EXPT(r_following_3,2)))*3600);  // Following erroring terms of a radius. 
	END_IF
(*
	IF ABS(r_following_3)> ABS(r_track_error[2]) THEN	
		r_following_33:=r_track_error[2];
	ELSE
		r_following_33:=r_following_33;
	END_IF
		IF ABS(r_following_33)>0.01 THEN
			r_following_33:=r_following_33/10;
		END_IF
	IF ABS(r_vel_EL)<0.0001 THEN
		r_following_3:=r_following_33;
	ELSE
		r_following_3:=r_following_33/p_covert_velocity_el;
	END_IF	
*)	
(*<<<<<<<<<<<<when finish all the points or the power is down,then reset the track_on>>>>>>>>>>>>>>>>>>>*)
	IF i_start=i_end OR b_remote_on_run=FALSE THEN
		 b_track_on:=FALSE;
	END_IF
(*<<<<<<<<<<<<<<<<<<<<<<<<<<<<stop the motion before tracking>>>>>>>>>>>>>>>>>>>*)
	IF r_rtrig_start_stop.Q THEN
		b_SCC_STOP:=TRUE;
	END_IF
	IF rtrig_track_on.Q=TRUE THEN
(*<<<<<<<<<<<<<<<<<<<<<<<<<<<<<<find the first point which can be caught up>>>>>>>>>>>>>>>>>>>>>>>>>>>*)
		//WHILE ABS(track_table[i_start].Azimuth-r_pos_az_v)/((track_table[i_start].MJD-lr_mjd_current)*86400-0.05)>2.9 OR (track_table[i_start].MJD-lr_mjd_current)*86400-0.05<0 DO
		test3:=ABS(track_table[i_start].Azimuth-r_pos_az_v)/((track_table[i_start].TAIoffset-lr_TAIoffset_current)-0.05)>2.9 OR (track_table[i_start].TAIoffset-lr_TAIoffset_current)-0.05<0;
		WHILE ABS(track_table[i_start].Azimuth-r_pos_az_v)/((track_table[i_start].TAIoffset-lr_TAIoffset_current)-0.05)>2.9 OR (track_table[i_start].TAIoffset-lr_TAIoffset_current)-0.05<0 DO
		//WHILE ABS(entry_buffer1[i_start].Azimuth-r_pos_az_v)/((entry_buffer1[i_start].MJD-lr_mjd_current)*86400-0.05)>2.9 DO
			IF i_start=i_end-3 THEN
				EXIT;
			ELSE
				i_start:=F_I_number(i_start+1);
			END_IF
		END_WHILE
		
		//WHILE ABS(track_table[i_start].Elevation-r_pos_el)/((track_table[i_start].MJD-lr_mjd_current)*86400-0.05)>0.8 OR (track_table[i_start].MJD-lr_mjd_current)*86400-0.05<0 DO
		test4:=ABS(track_table[i_start].Elevation-r_pos_el)/((track_table[i_start].TAIoffset-lr_TAIoffset_current)-0.05)>0.8 OR (track_table[i_start].TAIoffset-lr_TAIoffset_current)-0.05<0;
		WHILE ABS(track_table[i_start].Elevation-r_pos_el)/((track_table[i_start].TAIoffset-lr_TAIoffset_current)-0.05)>0.8 OR (track_table[i_start].TAIoffset-lr_TAIoffset_current)-0.05<0 DO	
		//WHILE ABS(entry_buffer1[i_start].Elevation-r_pos_motor3)/((entry_buffer1[i_start].MJD-lr_mjd_current)*86400-0.05)>1000 DO
			IF i_start=i_end-3 THEN
				EXIT;
			ELSE
				i_start:=F_I_number(i_start+1);
			END_IF
		END_WHILE
(*		WHILE ABS(entry_buffer1[i_start].FeedIndexer-r_pos_FI_v)/((entry_buffer1[i_start].MJD-lr_mjd_current)*86400-0.05)>2 OR (entry_buffer1[i_start].MJD-lr_mjd_current)*86400-0.05<0 DO
			IF i_start=i_end-3 THEN
				EXIT;
			ELSE
				i_start:=F_I_number(i_start+1);
			END_IF
		END_WHILE
*)

//		arAxisCtrl_gb[Drive3.AxisNo].Admin._OpMode.en := ModeCyclicVelocity; 
		b_write_el_vel:=TRUE;
		i_point_caught:=i_start;
		//i_caught_MJD1:=track_table[i_point_caught].MJD;
		 i_caught_TAIoffset1:=track_table[i_point_caught].TAIoffset;
		//i_caught_MJD2:=lr_MJD_current;
		i_caught_TAIoffset2:=lr_TAIoffset_current;
		r_start_az:=r_pos_az_v;
		r_caught_az:=track_table[i_point_caught].Azimuth;
		
(*if the first point which can be caught up is the last one£¬reset track_on*)
		IF i_start=i_end-3 THEN
			b_track_on:=FALSE;
		ELSE
			//track_table[F_I_number(i_start-1)].MJD:=lr_MJD_current+0.0000008;(*(69ms)after gunner change p41 from 0 to 100ms*)
			track_table[F_I_number(i_start-1)].TAIoffset:=lr_TAIoffset_current+0.069;(*(69ms)after gunner change p41 from 0 to 100ms*)
			track_table[F_I_number(i_start-1)].Azimuth:=r_pos_az_v;
			track_table[F_I_number(i_start-1)].elevation:=r_pos_el;
(*			entry_buffer1[F_I_number(i_start-1)].FeedIndexer:=r_pos_FI_v;  *)
		i_start:=F_I_number(i_start-1);
		r_write_position_az:=track_table[i_start].Azimuth;
		r_write_position_el:=track_table[i_start].Elevation;
(*		r_write_position_FI:=entry_buffer1[i_start].FeedIndexer;   *)
		r_last_position_az:=r_write_position_az;
		r_last_position_el:=r_write_position_el;
(*		r_last_position_FI:=r_write_position_FI;   *)
		b_signal_for_open:=TRUE;
		END_IF

	END_IF
(*when the position is all nearby the start point,open the channel for writing position to all axis*)
test5:=b_signal_for_open AND (ABS(r_pos_az_v-track_table[i_start].Azimuth)<0.001) AND (ABS(r_pos_el-track_table[i_start].Elevation)<0.001);
	IF b_signal_for_open AND (ABS(r_pos_az_v-track_table[i_start].Azimuth)<0.001) AND (ABS(r_pos_el-track_table[i_start].Elevation)<0.001) THEN
		b_open_channel_az:=TRUE;
//		b_start_cyclicvel:=TRUE;
//		b_open_channel_el:=TRUE;
(*		b_open_channel_FI:=TRUE;*)
		b_signal_for_open:=FALSE;
	END_IF
(*defind the variables for calculating the cubic fuction*)
		//t:=lr_MJD_current;
		//t1:=track_table[i_start].MJD;
		//t2:=track_table[F_I_number(i_start+1)].MJD;
		//t3:=track_table[F_I_number(i_start+2)].MJD;
		t:=lr_TAIoffset_current;
		t1:=track_table[i_start].TAIoffset;
		t2:=track_table[F_I_number(i_start+1)].TAIoffset;
		t3:=track_table[F_I_number(i_start+2)].TAIoffset;
		p1_az:=track_table[i_start].Azimuth;
		p2_az:=track_table[F_I_number(i_start+1)].Azimuth;
		p3_az:=track_table[F_I_number(i_start+2)].Azimuth;
		
		r_test1:=p1_az;
		r_test2:=p2_az;
		r_test3:=p3_az;
		
		p1_el:=track_table[i_start].elevation;
		p2_el:=track_table[F_I_number(i_start+1)].elevation;
		p3_el:=track_table[F_I_number(i_start+2)].elevation;		
(*		p1_FI:=entry_buffer1[i_start].FeedIndexer;
		p2_FI:=entry_buffer1[F_I_number(i_start+1)].FeedIndexer;
		p3_FI:=entry_buffer1[F_I_number(i_start+2)].FeedIndexer;
*)		
		//i_start;
		test_1:=F_I_number(i_start+1);
		test_2:=F_I_number(i_start+2);
(*construct the first cubic section by 2 points and 2 velocity*)
(*	IF	lr_MJD_current<entry_buffer1[i_point_caught].MJD AND lr_MJD_current>entry_buffer1[F_I_number(i_point_caught-1)].MJD THEN  *)
	//IF	lr_MJD_current<i_caught_MJD1 AND lr_MJD_current>i_caught_MJD2 THEN
test6:=lr_TAIoffset_current<i_caught_TAIoffset1 AND lr_TAIoffset_current>i_caught_TAIoffset2;
 IF	lr_TAIoffset_current<i_caught_TAIoffset1 AND lr_TAIoffset_current>i_caught_TAIoffset2 THEN	
	
		IF b_track_on THEN
			V_start_az:=(p3_az-p2_az)/(t3-t2);
			V_start_el:=(p3_el-p2_el)/(t3-t2);
(*			V_start_FI:=(p3_FI-p2_FI)/(t3-t2);  *)
			v0_az:=V_start_az;
			v0_el:=V_start_el;
(*			v0_FI:=V_start_FI;   *)
			b_test:=TRUE;
			b_start_to_compensate:=TRUE;

			a_az:=V_start_az/(t2-t1)/(t2-t1)-2*(p2_az-p1_az)/(t2-t1)/(t2-t1)/(t2-t1);
			b_az:=3*(p2_az-p1_az)/(t2-t1)/(t2-t1)-V_start_az/(t2-t1);
			a_el:=V_start_el/(t2-t1)/(t2-t1)-2*(p2_el-p1_el)/(t2-t1)/(t2-t1)/(t2-t1);
			b_el:=3*(p2_el-p1_el)/(t2-t1)/(t2-t1)-V_start_el/(t2-t1);
(*			a_FI:=V_start_FI/(t2-t1)/(t2-t1)-2*(p2_FI-p1_FI)/(t2-t1)/(t2-t1)/(t2-t1);
			b_FI:=3*(p2_FI-p1_FI)/(t2-t1)/(t2-t1)-V_start_FI/(t2-t1);
*)
			r_write_position_az:=a_az*(t-t1)*(t-t1)*(t-t1)+b_az*(t-t1)*(t-t1)+p1_az;
			r_write_position_el:=a_el*(t-t1)*(t-t1)*(t-t1)+b_el*(t-t1)*(t-t1)+p1_el;
(*			r_write_position_FI:=a_FI*(t-t1)*(t-t1)*(t-t1)+b_FI*(t-t1)*(t-t1)+p1_FI;   *)
		END_IF
	ELSE
		IF i_num_stack_left>2 THEN
			IF b_track_on THEN
(*<<<<<<<<<<<<<<<<<<<<<<<<<<<<<calculate the a and b in the function y=ax^3+bx^2+cx+d>>>>>>>>>>>>>>>>>>>>>>*)
(*y=a*(x-x1)^3+b*(x-x1)^2+c(x-x1)+d,   c=v0,  d=y1*)
			a_az:=((p3_az-p1_az)/(t3-t1)/(t3-t1)-(p2_az-p1_az)/(t2-t1)/(t2-t1)-v0_az/(t3-t1)+v0_az/(t2-t1))/(t3-t2);
			b_az:=((p3_az-p1_az)*(t2-t1)/(t3-t1)/(t3-t1)-(p2_az-p1_az)*(t3-t1)/(t2-t1)/(t2-t1)-v0_az*(t2-t1)/(t3-t1)+v0_az*(t3-t1)/(t2-t1))/(t2-t3);
			a_el:=((p3_el-p1_el)/(t3-t1)/(t3-t1)-(p2_el-p1_el)/(t2-t1)/(t2-t1)-v0_el/(t3-t1)+v0_el/(t2-t1))/(t3-t2);
			b_el:=((p3_el-p1_el)*(t2-t1)/(t3-t1)/(t3-t1)-(p2_el-p1_el)*(t3-t1)/(t2-t1)/(t2-t1)-v0_el*(t2-t1)/(t3-t1)+v0_el*(t3-t1)/(t2-t1))/(t2-t3);
(*			a_FI:=((p3_FI-p1_FI)/(t3-t1)/(t3-t1)-(p2_FI-p1_FI)/(t2-t1)/(t2-t1)-v0_FI/(t3-t1)+v0_FI/(t2-t1))/(t3-t2);
			b_FI:=((p3_FI-p1_FI)*(t2-t1)/(t3-t1)/(t3-t1)-(p2_FI-p1_FI)*(t3-t1)/(t2-t1)/(t2-t1)-v0_FI*(t2-t1)/(t3-t1)+v0_FI*(t3-t1)/(t2-t1))/(t2-t3);
*)
b_test:=FALSE;
			//IF lr_MJD_current>=track_table[i_start].MJD AND lr_MJD_current<=track_table[F_I_number(i_start+1)].MJD THEN
			test7:=lr_TAIoffset_current>=track_table[i_start].TAIoffset AND lr_TAIoffset_current<=track_table[F_I_number(i_start+1)].TAIoffset;
			IF lr_TAIoffset_current>=track_table[i_start].TAIoffset AND lr_TAIoffset_current<=track_table[F_I_number(i_start+1)].TAIoffset THEN
			
				r_write_position_az:=a_az*(t-t1)*(t-t1)*(t-t1)+b_az*(t-t1)*(t-t1)+v0_az*(t-t1)+p1_az;
				r_write_position_el:=a_el*(t-t1)*(t-t1)*(t-t1)+b_el*(t-t1)*(t-t1)+v0_el*(t-t1)+p1_el;
				r_cyclic_velocity_test:=(p2_el-p1_el)/(t2-t1)/86400;
				//r_cyclic_velocity_test:=(p2_el-p1_el)/(t2-t1);
				r_cyclic_velocity:=V0_el/86400;
				// r_cyclic_velocity:=V0_el;
(*				r_write_position_FI:=a_FI*(t-t1)*(t-t1)*(t-t1)+b_FI*(t-t1)*(t-t1)+v0_FI*(t-t1)+p1_FI;   *)
			END_IF
(*calculate the velocity of the last point*)
			//IF (lr_MJD_current-track_table[F_I_number(i_start+1)].MJD)*86400>=-0.002 AND (lr_MJD_current-track_table[F_I_number(i_start+1)].MJD)*86400<0 THEN
			test8:=(lr_TAIoffset_current-track_table[F_I_number(i_start+1)].TAIoffset)>=-0.002 AND (lr_TAIoffset_current-track_table[F_I_number(i_start+1)].TAIoffset)<0;
			IF (lr_TAIoffset_current-track_table[F_I_number(i_start+1)].TAIoffset)>=-0.002 AND (lr_TAIoffset_current-track_table[F_I_number(i_start+1)].TAIoffset)<0 THEN
				V0_az:=3*a_az*(t2-t1)*(t2-t1)+2*b_az*(t2-t1)+v0_az;
				V0_el:=3*a_el*(t2-t1)*(t2-t1)+2*b_el*(t2-t1)+v0_el;
(*				V0_FI:=3*a_FI*(t2-t1)*(t2-t1)+2*b_FI*(t2-t1)+v0_FI;    *)
			END_IF
			END_IF
		ELSE
(*<<<<<<<<<<<<<<<<<<<<<<<<run the last two points>>>>>>>>>>>>>>>>>>>>>>>>>>*)
			IF b_track_on THEN 
				//IF lr_MJD_current>=track_table[i_start].MJD AND lr_MJD_current<=track_table[F_I_number(i_start+1)].MJD THEN
				test9:= lr_TAIoffset_current>=track_table[i_start].TAIoffset AND lr_TAIoffset_current<=track_table[F_I_number(i_start+1)].TAIoffset;
				IF lr_TAIoffset_current>=track_table[i_start].TAIoffset AND lr_TAIoffset_current<=track_table[F_I_number(i_start+1)].TAIoffset THEN
				r_write_position_az:=(p2_az-p1_az)*(t-t1)/(t2-t1)+p1_az;
				r_write_position_el:=(p2_el-p1_el)*(t-t1)/(t2-t1)+p1_el;
(*				r_write_position_FI:=((p2_FI-p1_FI)*(t-t1)/(t2-t1)+p1_FI);     *)
				END_IF
			END_IF
		END_IF
	END_IF

	
IF b_start_to_compensate THEN
//	r_offset_el:=r_compensation_value_motor;
	r_write_position_az:=r_write_position_az+r_test_offset_az;
	r_write_position_el:=r_write_position_el+r_test_offset_el;
//	r_write_position_el:=r_write_position_el+r_offset_el;
END_IF
	
(*<<<<<<<<<<<<<<<<<<<<<<<<<limit the trajectory speed >>>>>>>>>>>>>>>>>>>>>>>>>*)
(*Because the program runs every 2ms,so wo can limit the position by the rule ¦¤y<v*¦¤t.*)
(*Azimuth trajectory speed limit is 5.1¡ã/s*)


		IF r_write_position_az-r_last_position_az>0.0031 THEN
				r_write_position_az:=r_last_position_az+0.0031;
				b_track_overspeed_az:=1;
			ELSIF r_write_position_az-r_last_position_az<-0.0031 THEN
				r_write_position_az:=r_last_position_az-0.0031;
				b_track_overspeed_az:=1;
			ELSE
				b_track_overspeed_az:=0;
			END_IF
(*Elevation trajectory speed limit is 1.05¡ã/s*)
			IF r_write_position_el-r_last_position_el>0.00091 THEN
				r_write_position_el:=r_last_position_el+0.00091;
				b_track_overspeed_el:=1;
			ELSIF r_write_position_el-r_last_position_el<-0.00091 THEN
				r_write_position_el:=r_last_position_el-0.00091;
				b_track_overspeed_el:=1;
			ELSE
				b_track_overspeed_el:=0;
			END_IF
(*
(*FeedIndexer trajectory speed limit is 2.1¡ã/s*)
			IF r_write_position_FI-r_last_position_FI>0.0042 THEN
				r_write_position_FI:=r_last_position_FI+0.0042;
				b_track_overspeed_FI:=1;
			ELSIF r_write_position_FI-r_last_position_FI<-0.0042 THEN
				r_write_position_FI:=r_last_position_FI-0.0042;
				b_track_overspeed_FI:=1;
			ELSE
				b_track_overspeed_FI:=0;
			END_IF
*)
			
			
(*register the velocity and position for calculate the speed limit and acceleration limit*)
			r_last_position_az:=r_write_position_az;
			r_last_position_el:=r_write_position_el;
(*			r_last_position_FI:=r_write_position_FI;   *)
(*<<<<<<<<<<<<<<<<<<<<<<<<close the cyclic channel and reset the track error>>>>>>>>>>>>>>>>>>>>>>>>>>*)
ELSE
(*close the cyclic channel*)
	b_open_channel_az:=FALSE;
	b_open_channel_el:=FALSE;
	b_start_to_compensate:=FALSE;
	r_compensation_value_motor:=0;
(*	b_open_channel_FI:=FALSE;  *)
(*reset the following error and so on*)
    r_write_position_el:= axisdata[8].rActualPosition_i;
	r_write_position_az:=  axisdata[7].rActualPosition_i;
	r_track_error[1]:=0;
	r_track_error[2]:=0;
	r_track_error[3]:=0;
	V0_az:=0;
	V0_el:=0;
	V_start_az:=0;
	V_start_el:=0;
	IF NOT(b_SCC_goto) AND NOT(b_track_on) THEN 
		r_following_1:=0.00;
		r_following_3:=0.00;
	END_IF
END_IF

 IF  b_test_offset_start THEN
	 	r_offset_t:=r_offset_t+0.001;
		test_t:=r_offset_t-r_offset_t1_acc-r_offset_t2_v;
 		(*****************AZ offset**********)
		r_az_offset_abs:=ABS(r_offset_az);
		r_offset_t1_acc:=r_az_offset_Vmax/r_az_offset_acc;
	 	r_offset_t3_dec:=r_az_offset_Vmax/r_az_offset_dec;
	 	l_offset_t1_acc:=0.5*r_az_offset_acc*r_offset_t1_acc*r_offset_t1_acc;
	 	l_offset_t3_dec:=0.5*r_az_offset_dec*r_offset_t3_dec*r_offset_t3_dec;
 		r_offset_t2_v:=(r_az_offset_abs-l_offset_t1_acc-l_offset_t3_dec)/r_az_offset_Vmax;
		l_offset_t2_v:=r_az_offset_Vmax*r_offset_t2_v;

			IF r_offset_t <=r_offset_t1_acc THEN
				r_test_offset_az_abs:=0.5*r_az_offset_acc*r_offset_t*r_offset_t;
			ELSIF r_offset_t1_acc<r_offset_t AND r_offset_t<(r_offset_t1_acc+r_offset_t2_v) THEN 
				r_test_offset_az_abs:=r_test_offset_az_abs+0.001*r_az_offset_Vmax;
			ELSIF (r_offset_t1_acc+r_offset_t2_v)<=r_offset_t AND r_offset_t<(r_offset_t1_acc+r_offset_t2_v+r_offset_t3_dec) THEN
				r_test_offset_az_abs:=l_offset_t1_acc+l_offset_t2_v+(r_offset_t-r_offset_t1_acc-r_offset_t2_v)*r_az_offset_Vmax-0.5*r_az_offset_dec*(r_offset_t-r_offset_t1_acc-r_offset_t2_v)*(r_offset_t-r_offset_t1_acc-r_offset_t2_v);
			ELSE 
				r_test_offset_az_abs:=r_az_offset_abs;
			END_IF

		IF r_test_offset_az_abs>=r_az_offset_abs THEN
			r_test_offset_az_abs:=r_az_offset_abs;
		END_IF
		IF r_offset_az<0 THEN
			r_test_offset_az:=-r_test_offset_az_abs;
		ELSE 
			r_test_offset_az:=r_test_offset_az_abs;
		END_IF
		r_test_offset_az:=r_offset_az_old+r_test_offset_az;
		
		
			(*****************EL offset**********)
		r_el_offset_abs:=ABS(r_offset_el);
		r_offset_t1_acc_el:=r_el_offset_Vmax/r_el_offset_acc;
	 	r_offset_t3_dec_el:=r_el_offset_Vmax/r_el_offset_dec;
	 	l_offset_t1_acc_el:=0.5*r_el_offset_acc*r_offset_t1_acc_el*r_offset_t1_acc_el;
	 	l_offset_t3_dec_el:=0.5*r_el_offset_dec*r_offset_t3_dec_el*r_offset_t3_dec_el;
 		r_offset_t2_v_el:=(r_el_offset_abs-l_offset_t1_acc_el-l_offset_t3_dec_el)/r_el_offset_Vmax;
		l_offset_t2_v_el:=r_el_offset_Vmax*r_offset_t2_v_el;

			IF r_offset_t <=r_offset_t1_acc_el THEN
				r_test_offset_el_abs:=0.5*r_el_offset_acc*r_offset_t*r_offset_t;
			ELSIF r_offset_t1_acc_el<r_offset_t AND r_offset_t<(r_offset_t1_acc_el+r_offset_t2_v_el) THEN 
				r_test_offset_el_abs:=r_test_offset_el_abs+0.001*r_el_offset_Vmax;
			ELSIF (r_offset_t1_acc_el+r_offset_t2_v_el)<=r_offset_t AND r_offset_t<(r_offset_t1_acc_el+r_offset_t2_v_el+r_offset_t3_dec_el) THEN
				r_test_offset_el_abs:=l_offset_t1_acc_el+l_offset_t2_v_el+(r_offset_t-r_offset_t1_acc_el-r_offset_t2_v_el)*r_el_offset_Vmax-0.5*r_el_offset_dec*(r_offset_t-r_offset_t1_acc_el-r_offset_t2_v_el)*(r_offset_t-r_offset_t1_acc_el-r_offset_t2_v_el);
			ELSE 
				r_test_offset_el_abs:=r_el_offset_abs;
			END_IF

		IF r_test_offset_el_abs>=r_el_offset_abs THEN
			r_test_offset_el_abs:=r_el_offset_abs;
		END_IF
		IF r_offset_el<0 THEN
			r_test_offset_el:=-r_test_offset_el_abs;
		ELSE 
			r_test_offset_el:=r_test_offset_el_abs;
		END_IF
		r_test_offset_el:=r_offset_el_old+r_test_offset_el;
    IF 	r_test_offset_el_abs=r_el_offset_abs AND r_test_offset_az_abs=r_az_offset_abs THEN 	
		b_test_offset_start:=FALSE;
		b_offset_running:=FALSE;
	END_IF
				
ELSE
	i_test_offset_count:=0;
	r_offset_t:=0;
	r_offset_az_old:=r_test_offset_az;
	r_offset_el_old:=r_test_offset_el;
END_IF


P_Track_cubic.A_StaticPM();
P_Track_cubic.A_AmbTempPM();
P_Track_cubic.A_DynamicPM();


Tracking.Status.p_desired_El:=r_write_position_el-Tracking.Status.act_statOffset_value_El/gc_lr_arcsec2deg;
Tracking.Status.p_desired_Az:=r_write_position_az-(Tracking.Status.act_statOffset_value_Xel/gc_lr_arcsec2deg)/COS(ML_degtorad(r_write_position_el));

IF b_track_on THEN 
r_write_position_az_out:=r_write_position_az-Pointing.Status.StaticPmCorrVal_Az/gc_lr_arcsec2deg-Pointing.Status.TiltCorrVal_Az/gc_lr_arcsec2deg-Pointing.Status.AmbTempCorrVal_Az/gc_lr_arcsec2deg;
r_write_position_el_out:=r_write_position_el-Pointing.Status.StaticPmCorrVal_El/gc_lr_arcsec2deg-Pointing.Status.TiltCorrVal_El/gc_lr_arcsec2deg-Pointing.Status.AmbTempCorrVal_El/gc_lr_arcsec2deg;
END_IF

IF gc_b_sim_on THEN 
	P_Track_cubic.A_Sim_track_function_blocks();
ELSE	
	P_Track_cubic.A_track_fuction_blocks();
END_IF

ACTION A_track_fuction_blocks:
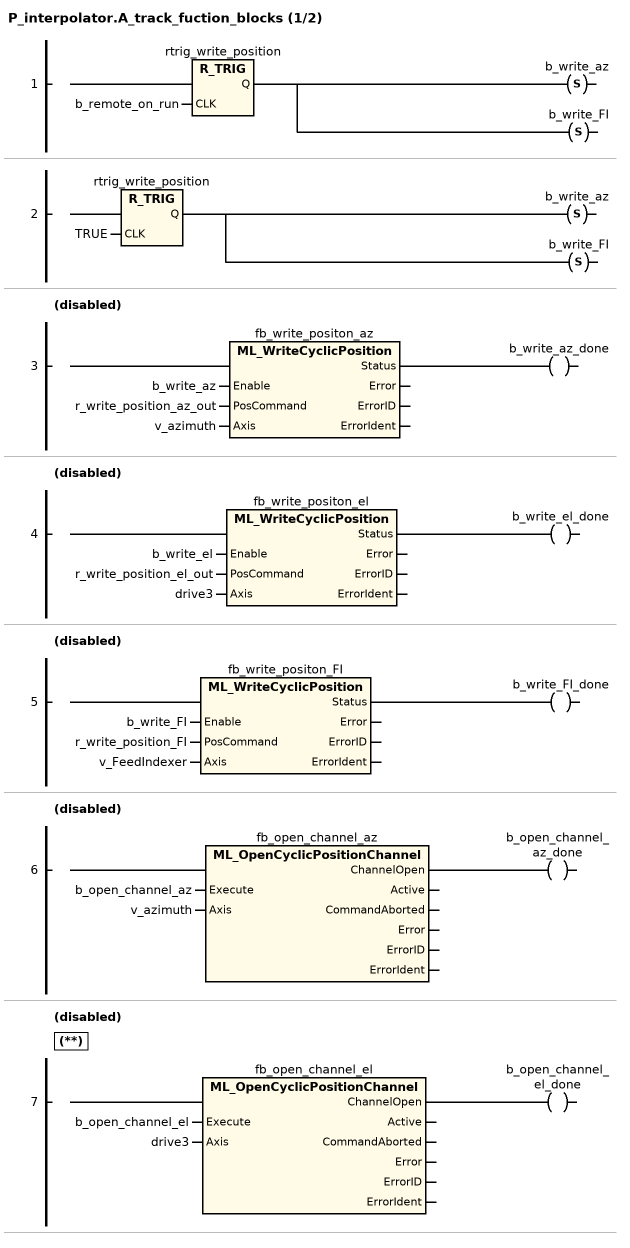
// NETWORK 1
rtrig_write_position(CLK := b_remote_on_run); // R_TRIG
b_write_az S= rtrig_write_position.Q;
b_write_FI S= rtrig_write_position.Q;

// NETWORK 2
rtrig_write_position(CLK := TRUE); // R_TRIG
b_write_az S= rtrig_write_position.Q;
b_write_FI S= rtrig_write_position.Q;

// NETWORK 3 (disabled)
// fb_write_positon_az(Enable := b_write_az, PosCommand := r_write_position_az_out, Axis := v_azimuth); // ML_WriteCyclicPosition
// b_write_az_done := fb_write_positon_az.Status;

// NETWORK 4 (disabled)
// fb_write_positon_el(Enable := b_write_el, PosCommand := r_write_position_el_out, Axis := drive3); // ML_WriteCyclicPosition
// b_write_el_done := fb_write_positon_el.Status;

// NETWORK 5 (disabled)
// fb_write_positon_FI(Enable := b_write_FI, PosCommand := r_write_position_FI, Axis := v_FeedIndexer); // ML_WriteCyclicPosition
// b_write_FI_done := fb_write_positon_FI.Status;

// NETWORK 6 (disabled)
// fb_open_channel_az(Execute := b_open_channel_az, Axis := v_azimuth); // ML_OpenCyclicPositionChannel
// b_open_channel_az_done := fb_open_channel_az.ChannelOpen;

// NETWORK 7 (disabled)
// label: (**)
// fb_open_channel_el(Execute := b_open_channel_el, Axis := drive3); // ML_OpenCyclicPositionChannel
// b_open_channel_el_done := fb_open_channel_el.ChannelOpen;

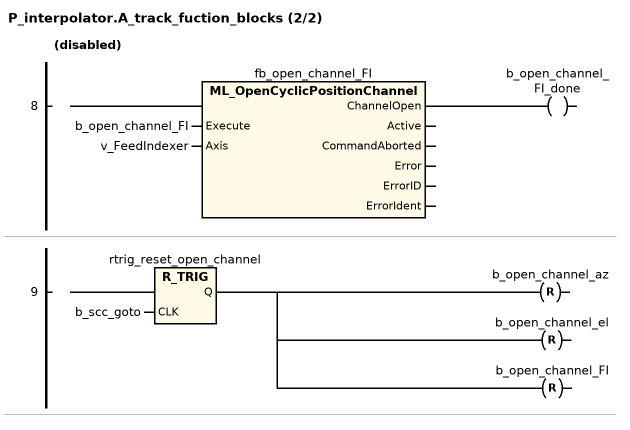
// NETWORK 8 (disabled)
// fb_open_channel_FI(Execute := b_open_channel_FI, Axis := v_FeedIndexer); // ML_OpenCyclicPositionChannel
// b_open_channel_FI_done := fb_open_channel_FI.ChannelOpen;

// NETWORK 9
rtrig_reset_open_channel(CLK := b_scc_goto); // R_TRIG
b_open_channel_az R= rtrig_reset_open_channel.Q;
b_open_channel_el R= rtrig_reset_open_channel.Q;
b_open_channel_FI R= rtrig_reset_open_channel.Q;
END_ACTION

ACTION A_StaticPM:
s_mp:= Pointing.StaticPmParameters[Pointing.Status.BandForCorr]; 

// Convert to Radians for trigonometric functions. 
Az_rad:= ML_degtorad(r_write_position_az);
IF r_write_position_el>= 85 THEN
	El_rad:= ML_degtorad(85);
ELSE
	El_rad:= ML_degtorad(r_write_position_el);	
END_IF

ABphi_rad:=ML_degtorad(s_mp.ABphi);

IF Pointing.Status.StaticCorrActive = 1 THEN 
	IF pointing.Status.TiltCorrActive = 1 THEN 
	// Calc Pointing correction with gravity tilt removed
	   TE := 0;
	ELSE 
	// Calc Pointing correction with gravity tilt
	   TE :=1;
    END_IF
	
	 Pointing.Status.StaticPmCorrVal_Az := ( -s_mp.IA - s_mp.CA/COS(El_rad) - s_mp.NPAE*TAN(El_rad) - s_mp.AN*SIN(Az_rad)*TAN(El_rad) - s_mp.AW*COS(Az_rad)*TAN(El_rad) + s_mp.ACEC*COS(Az_rad)
      - s_mp.ACES*SIN(Az_rad) - s_mp.ABA*SIN(ABphi_rad)*COS(2*Az_rad)*(1-TE) +   s_mp.ABA*COS(ABphi_rad)*SIN(2*Az_rad)*(1-TE) + Tracking.Status.act_statOffset_value_Xel/COS(El_rad) +
     (s_mp.AN0*SIN(Az_rad)*TAN(El_rad) + s_mp.AW0*COS(Az_rad)*TAN(El_rad))*TE);
	 
	(* Tiltmeter correction included in static pointing model.
       Pointing.Status.StaticPmCorrVal_Az :=  -s_mp.IA - s_mp.CA/COS(El) - s_mp.NPAE*TAN(El) - s_mp.AN*SIN(Az)*TAN(El) - s_mp.AW*COS(Az)*TAN(El) + s_mp.ACEC*COS(Az)
      - s_mp.ACES*SIN(Az) - s_mp.ABA*SIN(s_mp.ABphi)*COS(2*Az)*(1-TE) +   s_mp.ABA*COS(s_mp.ABphi)*SIN(2*Az)*(1-TE) + Tracking.Status.act_statOffset_value_Xel/COS(El) +
     (ΔAz_tiltmeter + s_mp.AN0*SIN(Az)*TAN(El) + s_mp.AW0*COS(Az)*TAN(El))*TE; *)
	
	Pointing.Status.StaticPmCorrVal_El := (s_mp.IE - s_mp.AN*COS(Az_rad) +s_mp.AW*SIN(Az_rad)+ s_mp.ECEC*COS(El_rad) + s_mp.ECES*SIN(El_rad) + s_mp.ABA*COS(ABphi_rad)*COS(2*Az_rad)*(1-TE) + s_mp.ABA*SIN(ABphi_rad)*SIN(2*Az_rad)*(1-TE) + 
    s_mp.HECE4*COS(4*El_rad) + s_mp.HESE4*SIN(4*El_rad) + s_mp.HECE8*COS(8*El_rad) + s_mp.HESE8*SIN(8*El_rad) + Tracking.Status.act_statOffset_value_El +
    (s_mp.AN0*COS(Az_rad) - s_mp.AW0*SIN(Az_rad))*TE);
	(*  Tiltmeter correction included in static pointing model.
	 Pointing.Status.StaticPmCorrVal_El := s_mp.IE - s_mp.AN*COS(Az) +s_mp.AW*SIN(Az)+ s_mp.ECEC*COS(El) + s_mp.ECES*SIN(El) + s_mp.ABA*COS(s_mp.ABphi)*COS(2*Az)*(1-TE) + s_mp.ABA*SIN(ABphi)*SIN(2*Az)*(1-TE) + 
    s_mp.HECE4*COS(4*El) + s_mp.HESE4*SIN(4*El) + s_mp.HECE8*COS(8*El) + s_mp.HESE8*SIN(8*El) + Tracking.Status.act_statOffset_value_El +
    (ΔEl_tiltmeter + s_mp.AN0*COS(Az) - s_mp.AW0*SIN(Az))*TE; *)
   
ELSE 
// No calculation of static model only offsets
   Pointing.Status.StaticPmCorrVal_Az := (Tracking.Status.act_statOffset_value_Xel/COS(El_rad));
   Pointing.Status.StaticPmCorrVal_El := Tracking.Status.act_statOffset_value_El;
END_IF


IF   ABS(Pointing.Status.StaticPmCorrVal_Az) > gc_lr_point_corr_error_lim OR  ABS(Pointing.Status.StaticPmCorrVal_El) > gc_lr_point_corr_error_lim THEN 
   Pointing.Status.StaticPmCorrVal_Az := 0; 
   Pointing.Status.StaticPmCorrVal_El := 0;
   Management.ErrorStatus.errPoint := 1; 
END_IF
END_ACTION

ACTION A_DynamicPM:
	IF Pointing.Status.TiltOne_On THEN 
    	Pointing.Status.TiltCorrVal_Az:= Pointing.Status.TiltYArcsec_One*TAN(El_rad); //El_rad is calculated in the Stati PM section 
		Pointing.Status.TiltCorrVal_El:= Pointing.Status.TiltXArcsec_One;
	ELSIF Pointing.Status.TiltTwo_On THEN
		Pointing.Status.TiltCorrVal_Az:= Pointing.Status.TiltYArcsec_One*TAN(El_rad);
		Pointing.Status.TiltCorrVal_El:= Pointing.Status.TiltXArcsec_One;
	ELSE
		Pointing.Status.TiltCorrVal_Az:= 0;
		Pointing.Status.TiltCorrVal_El:= 0;
	END_IF

//	Check velocity
IF  ABS(axisdata[1].rActualVelocity_i)>= gc_r_tilt_vel_limit_Az THEN 
	Pointing.Status.TiltCorrVal_Az:= 0;
    Pointing.Status.TiltCorrVal_El:= 0;
END_IF

// Check if the correction is with in limits 
// The behaviour if the correction is outside the limits still needs to be finalised
IF ABS(Pointing.Status.TiltCorrVal_Az)>= gc_lr_tilt_corr_limit_Az OR ABS(Pointing.Status.TiltCorrVal_El)>=gc_lr_tilt_corr_limit_El THEN 
	Pointing.Status.TiltCorrVal_Az:= gc_lr_tilt_corr_limit_Az;
    Pointing.Status.TiltCorrVal_El:= gc_lr_tilt_corr_limit_El;
END_IF
END_ACTION

ACTION A_AmbTempPM:
IF Pointing.Status.AmbTempCorrActive THEN 
	Pointing.Status.AmbTempCorrVal_Az:=0;
	Pointing.Status.AmbTempCorrVal_El:=0;
ELSE
	Pointing.Status.AmbTempCorrVal_Az:=0;
	Pointing.Status.AmbTempCorrVal_El:=0;
END_IF
END_ACTION

ACTION A_Sim_track_function_blocks:
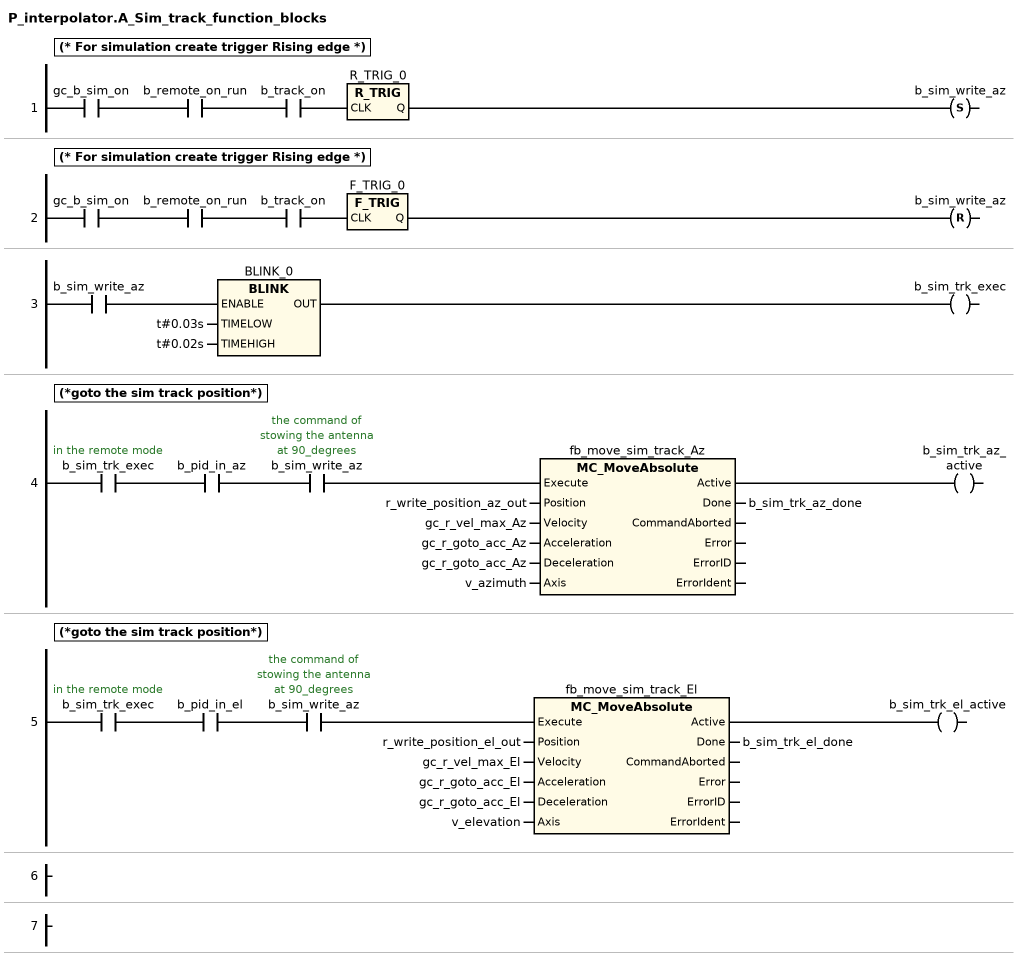
// NETWORK 1
// label: (* For simulation create trigger Rising edge *)
R_TRIG_0(CLK := gc_b_sim_on AND b_remote_on_run AND b_track_on); // R_TRIG
b_sim_write_az S= R_TRIG_0.Q;

// NETWORK 2
// label: (* For simulation create trigger Rising edge *)
F_TRIG_0(CLK := gc_b_sim_on AND b_remote_on_run AND b_track_on); // F_TRIG
b_sim_write_az R= F_TRIG_0.Q;

// NETWORK 3
BLINK_0(ENABLE := b_sim_write_az, TIMELOW := t#0.03s, TIMEHIGH := t#0.02s); // BLINK
b_sim_trk_exec := BLINK_0.OUT;

// NETWORK 4
//   fb_move_sim_track_Az: move the elevation to the fixed position
//   b_sim_trk_exec: in the remote mode
//   b_sim_write_az: the command of stowing the antenna at 90_degrees
//   v_azimuth: Virtual axis "v_elevation" with axis number 8
// label: (*goto the sim track position*)
fb_move_sim_track_Az(
    Execute := b_sim_trk_exec AND b_pid_in_az AND b_sim_write_az,
    Position := r_write_position_az_out,
    Velocity := gc_r_vel_max_Az,
    Acceleration := gc_r_goto_acc_Az,
    Deceleration := gc_r_goto_acc_Az,
    Axis := v_azimuth,
    Done => b_sim_trk_az_done); // MC_MoveAbsolute
b_sim_trk_az_active := fb_move_sim_track_Az.Active;

// NETWORK 5
//   fb_move_sim_track_El: move the elevation to the fixed position
//   b_sim_trk_exec: in the remote mode
//   b_sim_write_az: the command of stowing the antenna at 90_degrees
//   v_elevation: Virtual axis "v_elevation" with axis number 8
// label: (*goto the sim track position*)
fb_move_sim_track_El(
    Execute := b_sim_trk_exec AND b_pid_in_el AND b_sim_write_az,
    Position := r_write_position_el_out,
    Velocity := gc_r_vel_max_El,
    Acceleration := gc_r_goto_acc_El,
    Deceleration := gc_r_goto_acc_El,
    Axis := v_elevation,
    Done => b_sim_trk_el_done); // MC_MoveAbsolute
b_sim_trk_el_active := fb_move_sim_track_El.Active;

// NETWORK 6

// NETWORK 7
END_ACTION

END_PROGRAM

// IndraMotionMlc1/Application/AxisInterface/Visualizations/AxisModes/Axis_Overview
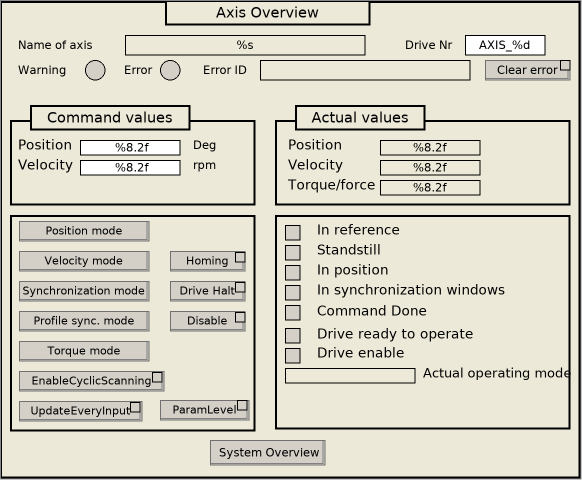
VISUALIZATION Axis_Overview  // 582x480
    Rectangle (0,1 580x477)
    Rectangle (15,35 110x20), "Name of axis"
    Rectangle (385,35 70x20), "Drive Nr"
    Rectangle (125,35 240x20), "%s", text variable: arAxisStatus_gb [VisuAxisNo].Admin.Name
    Ellipse (85,60 20x20), colour toggle: arAxisStatus_gb [VisuAxisNo].Diag.Warning
    Rectangle (15,60 70x20), "Warning"
    Ellipse (160,60 20x20), colour toggle: arAxisStatus_gb [VisuAxisNo].Diag.Error
    Rectangle (115,60 40x20), "Error"
    Rectangle (190,60 60x20), "Error ID"
    Rectangle (260,60 210x20), text list: 'ErrorIDCode', text index: arAxisStatus_gb [VisuAxisNo].Diag.ErrorID
    Button (485,60 85x20), "Clear error"
        tap arAxisCtrl_gb [VisuAxisNo].Admin.ClearError
    Rectangle (560,60 10x10), colour toggle: arAxisCtrl_gb [VisuAxisNo].Admin.ClearError
    Rectangle (165,0 205x25), "Axis Overview"
    Rectangle (10,215 245x216)
    Rectangle (10,120 245x85)
    Rectangle (275,120 295x85)
    Rectangle (295,105 130x25), "Actual values"
    Rectangle (15,135 80x20), "Position"
    Rectangle (285,135 80x20), "Position"
    Rectangle (285,155 80x20), "Velocity"
    Rectangle (285,175 100x20), "Torque/force"
    Rectangle (80,140 100x15), "%8.2f", text variable: arAxisCtrl_gb [VisuAxisNo].PosMode.Position
        OnMouseUp: write arAxisCtrl_gb [VisuAxisNo].PosMode.Position via 
    Rectangle (380,160 100x15), "%8.2f", text variable: AxisData[VisuAxisNo].rActualVelocity_i
    Rectangle (380,180 100x15), "%8.2f", text variable: AxisData[VisuAxisNo].rActualTorqueForce_i
    Rectangle (190,135 40x20), "Deg"
    Rectangle (190,155 40x20), "rpm"
    Rectangle (380,140 100x15), "%8.2f", text variable: AxisData[VisuAxisNo].rActualPosition_i
    Rectangle (80,160 100x15), "%8.2f", text variable: arAxisCtrl_gb [VisuAxisNo].VelMode.Velocity
        OnMouseUp: write arAxisCtrl_gb [VisuAxisNo].VelMode.Velocity via 
    Rectangle (15,155 70x20), "Velocity"
    Button (19,221 130x20), "Position mode"
        OnMouseUp:  Assign=Position_mode, Assign=Position_mode, Type=Assignment
    Button (19,251 130x20), "Velocity mode"
        OnMouseUp:  Assign=Velocity_mode, Assign=Velocity_mode, Type=Assignment
    Button (19,281 130x20), "Synchronization mode"
        OnMouseUp:  Assign=Synchronization_mode, Assign=Synchronization_mode, Type=Assignment
    Button (170,281 75x20), "Drive Halt"
        OnMouseUp: execute { arAxisCtrl_gb [VisuAxisNo].Admin._OpMode.en:=(ModeAh); }
    Rectangle (235,282 10x10), colour toggle: arAxisStatus_gb[VisuAxisNo].Admin._OpModeAck = ModeAH
    Rectangle (30,105 160x25), "Command values"
    Button (170,311 75x20), "Disable"
        OnMouseUp: execute { arAxisCtrl_gb [VisuAxisNo].Admin._OpMode.en:=(ModeAb); }
    Rectangle (235,312 10x10), colour toggle: arAxisStatus_gb[VisuAxisNo].Admin._OpModeAck = ModeAB
    Button (170,251 75x20), "Homing"
        OnMouseUp: execute { arAxisCtrl_gb [VisuAxisNo].Admin._OpMode.en:=(ModeHoming); }
    Rectangle (235,252 10x10), colour toggle: arAxisStatus_gb[VisuAxisNo].Admin._OpModeAck = ModeHoming
    Rectangle (275,215 295x214)
    Rectangle (285,265 15x15), colour toggle: (AxisData[VisuAxisNo].Axis_InPosition) <> 0
    Rectangle (285,285 15x15), colour toggle: (Axisdata[VisuAxisNo].Axis_InSynchron) <> 0
    Rectangle (314,240 100x20), "Standstill"
    Rectangle (314,260 100x20), "In position"
    Rectangle (314,280 250x20), "In synchronization windows"
    Rectangle (285,348 15x15), colour toggle: (AxisData[VisuAxisNo].Axis_Power) <> 0
    Rectangle (285,328 15x15), colour toggle: (AxisData[VisuAxisNo].Axis_InAb) <> 0
    Rectangle (314,343 170x20), "Drive enable"
    Rectangle (314,324 190x20), "Drive ready to operate"
    Rectangle (285,245 15x15), colour toggle: (AxisData[VisuAxisNo].Axis_Standstill) <> 0
    Rectangle (420,363 155x20), "Actual operating mode"
    Rectangle (285,225 15x15), colour toggle: (AxisData[VisuAxisNo].Axis_Homed) <> 0
    Rectangle (314,220 165x20), "In reference"
    Rectangle (285,368 130x15), text list: 'AxisMode', text index: arAxisStatus_gb [VisuAxisNo].Admin._OpModeAck
    Button (210,440 115x25), "System Overview"
        OnMouseUp:  Assign=System_Overview_All_Axis, Type=Assignment
    Rectangle (465,35 80x20), "AXIS_%d", text variable: VisuAxisNo
        OnMouseUp: write VisuAxisNo via 
    Button (19,311 130x20), "Profile sync. mode"
        OnMouseUp:  Assign=Profile_mode, Type=Assignment
    Button (160,400 89x20), "ParamLevel"
        toggle arAxisCtrl_gb[VisuAxisNo].Admin.ParamLevel
    Rectangle (237,400 10x10), colour toggle: arAxisStatus_gb[VisuAxisNo].Admin.ParamLevelAck = TRUE
    Button (19,371 145x20), "EnableCyclicScanning"
        toggle arAxisCtrl_gb[VisuAxisNo].Admin.EnableCyclicScanning
    Rectangle (152,372 10x10), colour toggle: arAxisCtrl_gb[VisuAxisNo].Admin.EnableCyclicScanning
    Button (19,401 123x20), "UpdateEveryInput"
        toggle arAxisCtrl_gb[VisuAxisNo].Admin.UpdateEveryInput
    Rectangle (130,402 10x10), colour toggle: arAxisCtrl_gb[VisuAxisNo].Admin.UpdateEveryInput
    Rectangle (285,305 15x15), colour toggle: (arAxisStatus_gb[VisuAxisNo].Admin.CmdDone) <> 0
    Rectangle (314,301 122x20), "Command Done"
    Button (19,341 130x20), "Torque mode"
        OnMouseUp:  Assign=Torque_mode, Type=Assignment
END_VISUALIZATION

// IndraMotionMlc1/Application/AxisInterface/Visualizations/AxisModes/Position_mode
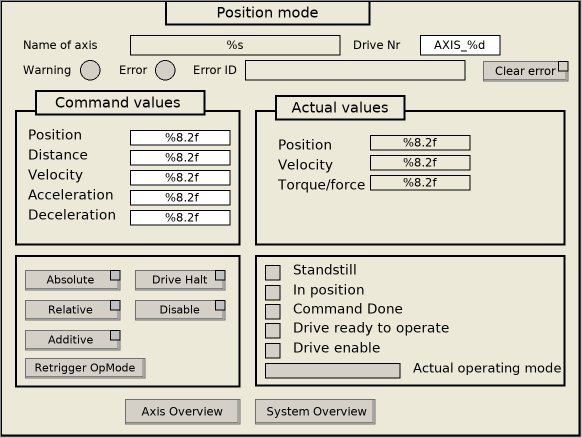
VISUALIZATION Position_mode  // 582x438
    Rectangle (0,0 580x436)
    Rectangle (15,255 225x132)
    Rectangle (165,0 205x25), "Position mode"
    Rectangle (15,110 225x135)
    Rectangle (35,90 170x25), "Command values"
    Rectangle (25,125 80x20), "Position"
    Rectangle (25,145 80x20), "Distance"
    Rectangle (25,165 80x20), "Velocity"
    Rectangle (130,150 100x15), "%8.2f", text variable: arAxisCtrl_gb [VisuAxisNo].PosMode.Distance
        OnMouseUp: write arAxisCtrl_gb [VisuAxisNo].PosMode.Distance via 
    Rectangle (130,170 100x15), "%8.2f", text variable: arAxisCtrl_gb [VisuAxisNo].PosMode.Velocity
        OnMouseUp: write arAxisCtrl_gb [VisuAxisNo].PosMode.Velocity via 
    Rectangle (130,130 100x15), "%8.2f", text variable: arAxisCtrl_gb [VisuAxisNo].PosMode.Position
        OnMouseUp: write arAxisCtrl_gb [VisuAxisNo].PosMode.Position via 
    Rectangle (130,190 100x15), "%8.2f", text variable: arAxisCtrl_gb [VisuAxisNo].PosMode.Acceleration
        OnMouseUp: write arAxisCtrl_gb [VisuAxisNo].PosMode.Acceleration via 
    Rectangle (25,185 100x20), "Acceleration"
    Rectangle (25,205 100x20), "Deceleration"
    Rectangle (130,210 100x15), "%8.2f", text variable: arAxisCtrl_gb [VisuAxisNo].PosMode.Deceleration
        OnMouseUp: write arAxisCtrl_gb [VisuAxisNo].PosMode.Deceleration via 
    Rectangle (255,110 310x135)
    Rectangle (275,95 130x25), "Actual values"
    Rectangle (275,135 80x20), "Position"
    Rectangle (275,155 80x20), "Velocity"
    Rectangle (275,175 100x20), "Torque/force"
    Rectangle (370,155 100x15), "%8.2f", text variable: AxisData[VisuAxisNo].rActualVelocity_i
    Rectangle (370,175 100x15), "%8.2f", text variable: AxisData[VisuAxisNo].rActualTorqueForce_i
    Rectangle (370,135 100x15), "%8.2f", text variable: AxisData[VisuAxisNo].rActualPosition_i
    Button (125,399 115x25), "Axis Overview"
        OnMouseUp:  Assign=Axis_Overview, Assign=Axis_Overview, Type=Assignment
    Rectangle (255,255 310x131)
    Rectangle (265,285 15x15), colour toggle: (AxisData[VisuAxisNo].Axis_InPosition) <> 0
    Rectangle (290,260 100x20), "Standstill"
    Rectangle (290,280 100x20), "In position"
    Rectangle (265,343 15x15), colour toggle: (AxisData[VisuAxisNo].Axis_Power) <> 0
    Rectangle (265,323 15x15), colour toggle: (AxisData[VisuAxisNo].Axis_InAb) <> 0
    Rectangle (290,338 170x20), "Drive enable"
    Rectangle (290,318 190x20), "Drive ready to operate"
    Rectangle (265,265 15x15), colour toggle: (AxisData[VisuAxisNo].Axis_Standstill) <> 0
    Button (25,270 95x20), "Absolute"
        OnMouseUp: execute { arAxisCtrl_gb [VisuAxisNo].Admin._OpMode.en:=(ModePosAbs); }
    Button (25,300 95x20), "Relative"
        OnMouseUp: execute { arAxisCtrl_gb [VisuAxisNo].Admin._OpMode.en:=(ModePosRel); }
    Rectangle (110,270 10x10), colour toggle: (arAxisStatus_gb[VisuAxisNo].Admin.MODE_POS_ABS) <> 0
    Rectangle (110,300 10x10), colour toggle: (arAxisStatus_gb[VisuAxisNo].Admin.MODE_POS_REL) <> 0
    Button (25,330 95x20), "Additive"
        OnMouseUp: execute { arAxisCtrl_gb [VisuAxisNo].Admin._OpMode.en:=(ModePosAdd); }
    Rectangle (110,330 10x10), colour toggle: (arAxisStatus_gb[VisuAxisNo].Admin.MODE_POS_ADD) <> 0
    Button (135,270 90x20), "Drive Halt"
        OnMouseUp: execute { arAxisCtrl_gb [VisuAxisNo].Admin._OpMode.en:=(ModeAh); }
    Rectangle (215,270 10x10), colour toggle: (arAxisStatus_gb[VisuAxisNo].Admin.MODE_AH) <> 0
    Button (135,300 90x20), "Disable"
        OnMouseUp: execute { arAxisCtrl_gb [VisuAxisNo].Admin._OpMode.en:=(ModeAb); }
    Rectangle (215,300 10x10), colour toggle: (arAxisStatus_gb[VisuAxisNo].Admin._OpModeAck = ModeAb) <> 0
    Rectangle (265,363 135x15), text list: 'AxisMode', text index: arAxisStatus_gb [VisuAxisNo].Admin._OpModeAck
    Rectangle (410,358 155x20), "Actual operating mode"
    Rectangle (20,35 110x20), "Name of axis"
    Rectangle (350,35 70x20), "Drive Nr"
    Rectangle (130,35 210x20), "%s", text variable: arAxisStatus_gb [VisuAxisNo].Admin.Name
    Ellipse (80,60 20x20), colour toggle: arAxisStatus_gb [VisuAxisNo].Diag.Warning
    Rectangle (20,60 70x20), "Warning"
    Ellipse (155,60 20x20), colour toggle: arAxisStatus_gb [VisuAxisNo].Diag.Error
    Rectangle (110,60 40x20), "Error"
    Rectangle (180,60 60x20), "Error ID"
    Rectangle (245,60 220x20), text list: 'ErrorIDCode', text index: arAxisStatus_gb [VisuAxisNo].Diag.ErrorID
    Button (255,399 120x25), "System Overview"
        OnMouseUp:  Assign=System_Overview_All_Axis, Assign=System_Overview_All_Axis, Type=Assignment
    Rectangle (420,35 80x20), "AXIS_%d", text variable: VisuAxisNo
        OnMouseUp: write VisuAxisNo via 
    Button (483,61 85x20), "Clear error"
        tap arAxisCtrl_gb [VisuAxisNo].Admin.ClearError
    Rectangle (558,61 10x10), colour toggle: arAxisCtrl_gb [VisuAxisNo].Admin.ClearError
    Button (25,358 120x20), "Retrigger OpMode"
        tap arAxisCtrl_gb[VisuAxisNo].Admin.RetriggerOpMode
    Rectangle (265,304 15x15), colour toggle: (arAxisStatus_gb[VisuAxisNo].Admin.CmdDone) <> 0
    Rectangle (290,299 122x20), "Command Done"
END_VISUALIZATION

// IndraMotionMlc1/Application/AxisInterface/Visualizations/AxisModes/Profile_mode
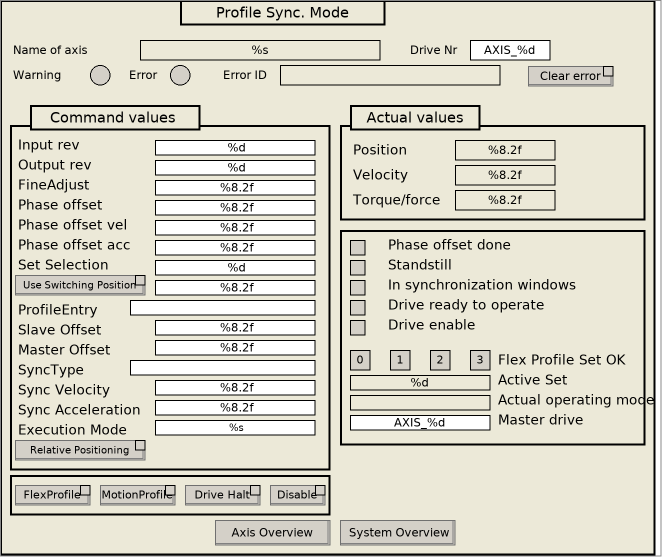
VISUALIZATION Profile_mode  // 662x557
    Rectangle (0,0 655x555)
    Rectangle (340,230 305x215)
    Rectangle (10,475 320x40)
    Button (100,485 75x20), "MotionProfile"
        OnMouseUp: execute { arAxisCtrl_gb [VisuAxisNo].Admin._OpMode.en:=(ModeSyncProfile); }
    Rectangle (180,0 205x25), "Profile Sync. Mode"
    Rectangle (10,125 320x345)
    Rectangle (30,105 170x25), "Command values"
    Rectangle (15,135 120x20), "Input rev"
    Rectangle (15,155 120x20), "Output rev"
    Rectangle (15,175 120x20), "FineAdjust"
    Rectangle (155,160 160x15), "%d", text variable: arAxisCtrl_gb [VisuAxisNo].SyncMode.OutputRevolution
        OnMouseUp: write arAxisCtrl_gb [VisuAxisNo].SyncMode.OutputRevolution via 
    Rectangle (155,180 160x15), "%8.2f", text variable: arAxisCtrl_gb [VisuAxisNo].SyncMode.FineAdjust
        OnMouseUp: write arAxisCtrl_gb [VisuAxisNo].SyncMode.FineAdjust via 
    Rectangle (155,140 160x15), "%d", text variable: arAxisCtrl_gb [VisuAxisNo].SyncMode.InputRevolution
        OnMouseUp: write arAxisCtrl_gb [VisuAxisNo].SyncMode.InputRevolution via 
    Rectangle (15,195 120x20), "Phase offset"
    Rectangle (155,200 160x15), "%8.2f", text variable: arAxisCtrl_gb [VisuAxisNo].SyncMode.PhaseOffset
        OnMouseUp: write arAxisCtrl_gb [VisuAxisNo].SyncMode.PhaseOffset via 
    Rectangle (155,220 160x15), "%8.2f", text variable: arAxisCtrl_gb [VisuAxisNo].SyncMode.PhaseOffsetVel
        OnMouseUp: write arAxisCtrl_gb [VisuAxisNo].SyncMode.PhaseOffsetVel via 
    Rectangle (15,215 140x20), "Phase offset vel"
    Rectangle (15,235 140x20), "Phase offset acc"
    Rectangle (155,240 160x15), "%8.2f", text variable: arAxisCtrl_gb [VisuAxisNo].SyncMode.PhaseOffsetAcc
        OnMouseUp: write arAxisCtrl_gb [VisuAxisNo].SyncMode.PhaseOffsetAcc via 
    Rectangle (340,125 305x95)
    Rectangle (350,105 130x25), "Actual values"
    Rectangle (350,140 100x20), "Position"
    Rectangle (350,165 100x20), "Velocity"
    Rectangle (350,190 110x20), "Torque/force"
    Rectangle (455,165 100x20), "%8.2f", text variable: AxisData[VisuAxisNo].rActualVelocity_i
    Rectangle (455,190 100x20), "%8.2f", text variable: AxisData[VisuAxisNo].rActualTorqueForce_i
    Rectangle (455,140 100x20), "%8.2f", text variable: AxisData[VisuAxisNo].rActualPosition_i
    Button (15,485 75x20), "FlexProfile"
        OnMouseUp: execute { arAxisCtrl_gb [VisuAxisNo].Admin._OpMode.en:=(ModeFlexProfile); }
    Rectangle (80,485 10x10), colour toggle: (arAxisStatus_gb[VisuAxisNo].Admin.MODE_FLEX_PROFILE) <> 0
    Rectangle (350,280 15x15), colour toggle: (AxisData[VisuAxisNo].Axis_InSynchron) <> 0
    Rectangle (385,255 100x20), "Standstill"
    Rectangle (385,275 240x20), "In synchronization windows"
    Rectangle (350,320 15x15), colour toggle: (AxisData[VisuAxisNo].Axis_Power) <> 0
    Rectangle (350,300 15x15), colour toggle: (AxisData[VisuAxisNo].Axis_InAb) <> 0
    Rectangle (385,295 190x20), "Drive ready to operate"
    Rectangle (350,260 15x15), colour toggle: (AxisData[VisuAxisNo].Axis_Standstill) <> 0
    Button (185,485 75x20), "Drive Halt"
        OnMouseUp: execute { arAxisCtrl_gb [VisuAxisNo].Admin._OpMode.en:=(ModeAh); }
    Rectangle (250,485 10x10), colour toggle: (arAxisStatus_gb[VisuAxisNo].Admin.MODE_AH) <> 0
    Button (270,485 55x20), "Disable"
        OnMouseUp: execute { arAxisCtrl_gb [VisuAxisNo].Admin._OpMode.en:=(ModeAb); }
    Rectangle (315,485 10x10), colour toggle: (arAxisStatus_gb[VisuAxisNo].Admin._OpModeAck = ModeAb) <> 0
    Rectangle (350,240 15x15), colour toggle: arAxisStatus_gb [VisuAxisNo].SyncMode.PhasingSlaveDone
    Rectangle (385,235 250x20), "Phase offset done"
    Rectangle (10,40 120x20), "Name of axis"
    Rectangle (390,40 70x20), "Drive Nr"
    Rectangle (140,40 240x20), "%s", text variable: arAxisStatus_gb [VisuAxisNo].Admin.Name
    Ellipse (90,65 20x20), colour toggle: arAxisStatus_gb [VisuAxisNo].Diag.Warning
    Rectangle (10,65 70x20), "Warning"
    Ellipse (170,65 20x20), colour toggle: arAxisStatus_gb [VisuAxisNo].Diag.Error
    Rectangle (120,65 40x20), "Error"
    Rectangle (200,65 70x20), "Error ID"
    Rectangle (280,65 220x20), text list: 'ErrorIDCode', text index: arAxisStatus_gb [VisuAxisNo].Diag.ErrorID
    Button (215,520 115x25), "Axis Overview"
        OnMouseUp:  Assign=Axis_Overview, Assign=Axis_Overview, Type=Assignment
    Button (340,520 115x25), "System Overview"
        OnMouseUp:  Assign=System_Overview_All_Axis, Assign=System_Overview_All_Axis, Type=Assignment
    Rectangle (385,315 170x20), "Drive enable"
    Rectangle (470,40 80x20), "AXIS_%d", text variable: VisuAxisNo
        OnMouseUp: write VisuAxisNo via 
    Rectangle (350,415 140x15), "AXIS_%d", text variable: arAxisCtrl_gb [VisuAxisNo].SyncMode.Master.AxisNo
        OnMouseUp: write arAxisCtrl_gb [VisuAxisNo].SyncMode.Master.AxisNo via 
    Rectangle (495,410 100x20), "Master drive"
    Rectangle (350,395 140x15), text list: 'AxisMode', text index: arAxisStatus_gb [VisuAxisNo].Admin._OpModeAck
    Rectangle (495,390 165x20), "Actual operating mode"
    Rectangle (15,255 140x20), "Set Selection"
    Rectangle (155,260 160x15), "%d", text variable: arAxisCtrl_gb [VisuAxisNo].SyncMode.Profile.SetSelection
        OnMouseUp: write arAxisCtrl_gb [VisuAxisNo].SyncMode.Profile.SetSelection via 
    Button (15,440 130x20), "Relative Positioning"
        toggle arAxisCtrl_gb [VisuAxisNo].SyncMode.Profile.RelativePositioning
    Rectangle (165,485 10x10), colour toggle: (arAxisStatus_gb[VisuAxisNo].Admin.MODE_SYNC_PROFILE) <> 0
    Rectangle (135,440 10x10), colour toggle: (arAxisCtrl_gb[VisuAxisNo].SyncMode.Profile.RelativePositioning) <> 0
    Button (15,275 130x20), "Use Switching Position"
        toggle arAxisCtrl_gb [VisuAxisNo].SyncMode.Profile.UseSwitchingPosition
    Rectangle (155,280 160x15), "%8.2f", text variable: arAxisCtrl_gb [VisuAxisNo].SyncMode.Profile.SwitchingPosition
        OnMouseUp: write arAxisCtrl_gb [VisuAxisNo].SyncMode.Profile.SwitchingPosition via 
    Rectangle (130,300 185x15), text list: 'ProfileEntry', text index: arAxisCtrl_gb [VisuAxisNo].SyncMode.Profile.ProfileEntry
        OnMouseUp: write arAxisCtrl_gb [VisuAxisNo].SyncMode.Profile.ProfileEntry via 
    Rectangle (155,320 160x15), "%8.2f", text variable: arAxisCtrl_gb [VisuAxisNo].SyncMode.Profile.SlaveOffset
        OnMouseUp: write arAxisCtrl_gb [VisuAxisNo].SyncMode.Profile.SlaveOffset via 
    Rectangle (155,340 160x15), "%8.2f", text variable: arAxisCtrl_gb [VisuAxisNo].SyncMode.Profile.MasterOffset
        OnMouseUp: write arAxisCtrl_gb [VisuAxisNo].SyncMode.Profile.MasterOffset via 
    Rectangle (15,300 140x20), "ProfileEntry"
    Rectangle (15,320 140x20), "Slave Offset"
    Rectangle (15,340 140x20), "Master Offset"
    Rectangle (130,360 185x15), text list: 'SyncType', text index: arAxisCtrl_gb [VisuAxisNo].SyncMode.Profile.SyncType
        OnMouseUp: write arAxisCtrl_gb [VisuAxisNo].SyncMode.Profile.SyncType via 
    Rectangle (155,380 160x15), "%8.2f", text variable: arAxisCtrl_gb [VisuAxisNo].SyncMode.SyncVelocity
        OnMouseUp: write arAxisCtrl_gb [VisuAxisNo].SyncMode.SyncVelocity via Edit
    Rectangle (155,400 160x15), "%8.2f", text variable: arAxisCtrl_gb [VisuAxisNo].SyncMode.SyncAcceleration
        OnMouseUp: write arAxisCtrl_gb [VisuAxisNo].SyncMode.SyncAcceleration via Edit
    Rectangle (155,420 160x15), "%s", text list: 'ExecutionMode', text index: arAxisCtrl_gb [VisuAxisNo].SyncMode.Profile.ExecutionMode
        OnMouseUp: write arAxisCtrl_gb [VisuAxisNo].SyncMode.Profile.ExecutionMode via 
    Rectangle (15,360 140x20), "SyncType"
    Rectangle (15,380 140x20), "Sync Velocity"
    Rectangle (15,400 140x20), "Sync Acceleration"
    Rectangle (15,420 140x20), "Execution Mode"
    Rectangle (135,275 10x10), colour toggle: (arAxisCtrl_gb[VisuAxisNo].SyncMode.Profile.UseSwitchingPosition) <> 0
    Rectangle (350,375 140x15), "%d", text variable: arAxisStatus_gb [VisuAxisNo].SyncMode.ProfileActiveSet
    Rectangle (495,370 165x20), "Active Set"
    Rectangle (350,350 20x20), "0", colour toggle: (AxisData[VisuAxisNo].FlexProfil_Set0_Ok) <> 0
    Rectangle (390,350 20x20), "1", colour toggle: (AxisData[VisuAxisNo].FlexProfil_Set1_Ok) <> 0
    Rectangle (430,350 20x20), "2", colour toggle: (AxisData[VisuAxisNo].FlexProfil_Set2_Ok) <> 0
    Rectangle (470,350 20x20), "3", colour toggle: (AxisData[VisuAxisNo].FlexProfil_Set3_Ok) <> 0
    Rectangle (495,350 130x20), "Flex Profile Set OK"
    Button (528,66 85x20), "Clear error"
        tap arAxisCtrl_gb [VisuAxisNo].Admin.ClearError
    Rectangle (603,66 10x10), colour toggle: arAxisCtrl_gb [VisuAxisNo].Admin.ClearError
END_VISUALIZATION

// IndraMotionMlc1/Application/AxisInterface/Visualizations/AxisModes/Synchronization_mode
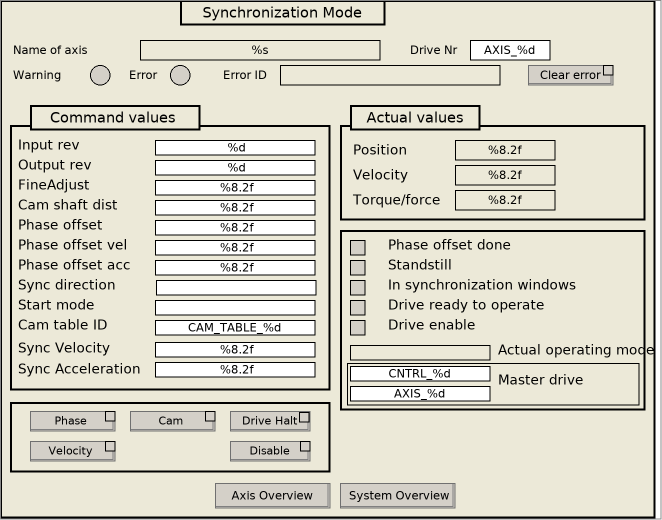
VISUALIZATION Synchronization_mode  // 662x520
    Rectangle (10,360 320x70)
    Rectangle (0,0 655x518)
    Rectangle (340,230 305x180)
    Rectangle (10,402 320x70)
    Rectangle (180,0 205x25), "Synchronization Mode"
    Rectangle (10,125 320x265)
    Rectangle (30,105 170x25), "Command values"
    Rectangle (15,135 120x20), "Input rev"
    Rectangle (15,155 120x20), "Output rev"
    Rectangle (15,175 120x20), "FineAdjust"
    Rectangle (155,160 160x15), "%d", text variable: arAxisCtrl_gb [VisuAxisNo].SyncMode.OutputRevolution
        OnMouseUp: write arAxisCtrl_gb [VisuAxisNo].SyncMode.OutputRevolution via 
    Rectangle (155,180 160x15), "%8.2f", text variable: arAxisCtrl_gb [VisuAxisNo].SyncMode.FineAdjust
        OnMouseUp: write arAxisCtrl_gb [VisuAxisNo].SyncMode.FineAdjust via 
    Rectangle (155,140 160x15), "%d", text variable: arAxisCtrl_gb [VisuAxisNo].SyncMode.InputRevolution
        OnMouseUp: write arAxisCtrl_gb [VisuAxisNo].SyncMode.InputRevolution via 
    Rectangle (155,200 160x15), "%8.2f", text variable: arAxisCtrl_gb [VisuAxisNo].SyncMode.CamShaftDistance
        OnMouseUp: write arAxisCtrl_gb [VisuAxisNo].SyncMode.CamShaftDistance via 
    Rectangle (15,195 120x20), "Cam shaft dist"
    Rectangle (15,215 120x20), "Phase offset"
    Rectangle (155,220 160x15), "%8.2f", text variable: arAxisCtrl_gb [VisuAxisNo].SyncMode.PhaseOffset
        OnMouseUp: write arAxisCtrl_gb [VisuAxisNo].SyncMode.PhaseOffset via 
    Rectangle (155,240 160x15), "%8.2f", text variable: arAxisCtrl_gb [VisuAxisNo].SyncMode.PhaseOffsetVel
        OnMouseUp: write arAxisCtrl_gb [VisuAxisNo].SyncMode.PhaseOffsetVel via 
    Rectangle (15,235 140x20), "Phase offset vel"
    Rectangle (15,255 140x20), "Phase offset acc"
    Rectangle (155,260 160x15), "%8.2f", text variable: arAxisCtrl_gb [VisuAxisNo].SyncMode.PhaseOffsetAcc
        OnMouseUp: write arAxisCtrl_gb [VisuAxisNo].SyncMode.PhaseOffsetAcc via 
    Rectangle (156,280 160x15), text list: 'SyncDirection', text index: arAxisCtrl_gb [VisuAxisNo].SyncMode.SyncDirection
        OnMouseUp: write arAxisCtrl_gb [VisuAxisNo].SyncMode.SyncDirection via 
    Rectangle (15,275 120x20), "Sync direction"
    Rectangle (15,295 120x20), "Start mode"
    Rectangle (155,300 160x15), text list: 'StartMode', text index: arAxisCtrl_gb [VisuAxisNo].SyncMode.StartMode
        OnMouseUp: write arAxisCtrl_gb [VisuAxisNo].SyncMode.StartMode via 
    Rectangle (155,320 160x15), "CAM_TABLE_%d", text variable: arAxisCtrl_gb [VisuAxisNo].SyncMode.CamTableID
        OnMouseUp: write arAxisCtrl_gb [VisuAxisNo].SyncMode.CamTableID via 
    Rectangle (15,315 120x20), "Cam table ID"
    Rectangle (340,125 305x95)
    Rectangle (350,105 130x25), "Actual values"
    Rectangle (350,140 100x20), "Position"
    Rectangle (350,165 100x20), "Velocity"
    Rectangle (350,190 110x20), "Torque/force"
    Rectangle (455,165 100x20), "%8.2f", text variable: AxisData[VisuAxisNo].rActualVelocity_i
    Rectangle (455,190 100x20), "%8.2f", text variable: AxisData[VisuAxisNo].rActualTorqueForce_i
    Rectangle (455,140 100x20), "%8.2f", text variable: AxisData[VisuAxisNo].rActualPosition_i
    Button (30,411 85x20), "Phase"
        OnMouseUp: execute { arAxisCtrl_gb [VisuAxisNo].Admin._OpMode.en:=(ModeSyncPhase); }
    Rectangle (105,411 10x10), colour toggle: (arAxisStatus_gb[VisuAxisNo].Admin.MODE_SYNC_PHASE) <> 0
    Button (30,441 85x20), "Velocity"
        OnMouseUp: execute { arAxisCtrl_gb [VisuAxisNo].Admin._OpMode.en:=(ModeSyncVel); }
    Rectangle (105,441 10x10), colour toggle: (arAxisStatus_gb[VisuAxisNo].Admin.MODE_SYNC_VEL) <> 0
    Button (130,411 85x20), "Cam"
        OnMouseUp: execute { arAxisCtrl_gb [VisuAxisNo].Admin._OpMode.en:=(ModeSyncCam); }
    Rectangle (205,411 10x10), colour toggle: (arAxisStatus_gb[VisuAxisNo].Admin.MODE_SYNC_CAM) <> 0
    Rectangle (350,280 15x15), colour toggle: (AxisData[VisuAxisNo].Axis_InSynchron) <> 0
    Rectangle (385,255 100x20), "Standstill"
    Rectangle (385,275 240x20), "In synchronization windows"
    Rectangle (350,320 15x15), colour toggle: (AxisData[VisuAxisNo].Axis_Power) <> 0
    Rectangle (350,300 15x15), colour toggle: (AxisData[VisuAxisNo].Axis_InAb) <> 0
    Rectangle (385,295 190x20), "Drive ready to operate"
    Rectangle (350,260 15x15), colour toggle: (AxisData[VisuAxisNo].Axis_Standstill) <> 0
    Button (230,411 80x20), "Drive Halt"
        OnMouseUp: execute { arAxisCtrl_gb [VisuAxisNo].Admin._OpMode.en:=(ModeAh); }
    Button (230,441 80x20), "Disable"
        OnMouseUp: execute { arAxisCtrl_gb [VisuAxisNo].Admin._OpMode.en:=(ModeAb); }
    Rectangle (300,441 10x10), colour toggle: (arAxisStatus_gb[VisuAxisNo].Admin._OpModeAck = ModeAb) <> 0
    Rectangle (350,240 15x15), colour toggle: arAxisStatus_gb [VisuAxisNo].SyncMode.PhasingSlaveDone
    Rectangle (385,235 250x20), "Phase offset done"
    Rectangle (10,40 120x20), "Name of axis"
    Rectangle (390,40 70x20), "Drive Nr"
    Rectangle (140,40 240x20), "%s", text variable: arAxisStatus_gb [VisuAxisNo].Admin.Name
    Ellipse (90,65 20x20), colour toggle: arAxisStatus_gb [VisuAxisNo].Diag.Warning
    Rectangle (10,65 70x20), "Warning"
    Ellipse (170,65 20x20), colour toggle: arAxisStatus_gb [VisuAxisNo].Diag.Error
    Rectangle (120,65 40x20), "Error"
    Rectangle (200,65 70x20), "Error ID"
    Rectangle (280,65 220x20), text list: 'ErrorIDCode', text index: arAxisStatus_gb [VisuAxisNo].Diag.ErrorID
    Button (215,483 115x25), "Axis Overview"
        OnMouseUp:  Assign=Axis_Overview, Assign=Axis_Overview, Type=Assignment
    Button (340,483 115x25), "System Overview"
        OnMouseUp:  Assign=System_Overview_All_Axis, Assign=System_Overview_All_Axis, Type=Assignment
    Rectangle (385,315 170x20), "Drive enable"
    Rectangle (470,40 80x20), "AXIS_%d", text variable: VisuAxisNo
        OnMouseUp: write VisuAxisNo via 
    Rectangle (350,366 140x15), "CNTRL_%d", text variable: arAxisCtrl_gb [VisuAxisNo].SyncMode.Master.CntrlNo
        OnMouseUp: write arAxisCtrl_gb [VisuAxisNo].SyncMode.Master.CntrlNo via Default
    Rectangle (495,370 100x20), "Master drive"
    Rectangle (350,345 140x15), text list: 'AxisMode', text index: arAxisStatus_gb [VisuAxisNo].Admin._OpModeAck
    Rectangle (495,340 165x20), "Actual operating mode"
    Rectangle (155,342 160x15), "%8.2f", text variable: arAxisCtrl_gb [VisuAxisNo].SyncMode.SyncVelocity
        OnMouseUp: write arAxisCtrl_gb [VisuAxisNo].SyncMode.SyncVelocity via Edit
    Rectangle (155,362 160x15), "%8.2f", text variable: arAxisCtrl_gb [VisuAxisNo].SyncMode.SyncAcceleration
        OnMouseUp: write arAxisCtrl_gb [VisuAxisNo].SyncMode.SyncAcceleration via Edit
    Rectangle (15,338 140x20), "Sync Velocity"
    Rectangle (15,359 140x20), "Sync Acceleration"
    Button (528,65 85x20), "Clear error"
        tap arAxisCtrl_gb [VisuAxisNo].Admin.ClearError
    Rectangle (603,65 10x10), colour toggle: arAxisCtrl_gb [VisuAxisNo].Admin.ClearError
    Rectangle (299,412 10x10), colour toggle: (arAxisStatus_gb[VisuAxisNo].Admin.MODE_AH) <> 0
    Rectangle (350,386 140x15), "AXIS_%d", text variable: arAxisCtrl_gb [VisuAxisNo].SyncMode.Master.AxisNo
        OnMouseUp: write arAxisCtrl_gb [VisuAxisNo].SyncMode.Master.AxisNo via 
    Rectangle (347,363 292x42)
END_VISUALIZATION

// IndraMotionMlc1/Application/AxisInterface/Visualizations/AxisModes/Torque_mode
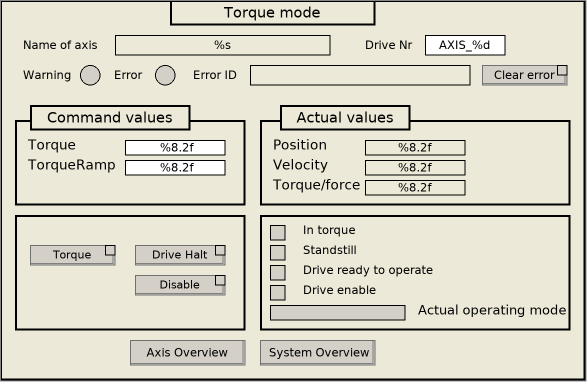
VISUALIZATION Torque_mode  // 587x382
    Rectangle (0,0 585x380)
    Rectangle (15,215 230x115)
    Rectangle (15,120 230x85)
    Rectangle (30,105 160x25), "Command values"
    Rectangle (25,135 80x20), "Torque"
    Rectangle (25,155 100x20), "TorqueRamp"
    Rectangle (125,160 100x15), "%8.2f", text variable: arAxisCtrl_gb [VisuAxisNo].TorqueMode.TorqueRamp
        OnMouseUp: write arAxisCtrl_gb [VisuAxisNo].TorqueMode.TorqueRamp via Edit
    Rectangle (125,140 100x15), "%8.2f", text variable: arAxisCtrl_gb [VisuAxisNo].TorqueMode.Torque
        OnMouseUp: write arAxisCtrl_gb [VisuAxisNo].TorqueMode.Torque via Edit
    Rectangle (260,120 310x85)
    Rectangle (280,105 130x25), "Actual values"
    Rectangle (270,135 70x20), "Position"
    Rectangle (270,155 75x20), "Velocity"
    Rectangle (270,175 90x20), "Torque/force"
    Rectangle (365,160 100x15), "%8.2f", text variable: AxisData[VisuAxisNo].rActualVelocity_i
    Rectangle (365,180 100x15), "%8.2f", text variable: AxisData[VisuAxisNo].rActualTorqueForce_i
    Rectangle (365,140 100x15), "%8.2f", text variable: AxisData[VisuAxisNo].rActualPosition_i
    Rectangle (170,0 205x25), "Torque mode"
    Button (30,245 85x20), "Torque"
        OnMouseUp: execute { arAxisCtrl_gb[VisuAxisNo].Admin._OpMode.en:=(ModeTorque); }
    Rectangle (105,245 10x10), colour toggle: arAxisStatus_gb[VisuAxisNo].Admin._OpModeAck = ModeTorque
    Rectangle (260,215 310x115)
    Rectangle (300,240 100x20), "Standstill"
    Rectangle (270,285 15x15), colour toggle: (AxisData[VisuAxisNo].Axis_Power) <> 0
    Rectangle (270,265 15x15), colour toggle: (AxisData[VisuAxisNo].Axis_InAb) <> 0
    Rectangle (300,280 170x20), "Drive enable"
    Rectangle (300,260 190x20), "Drive ready to operate"
    Rectangle (270,245 15x15), colour toggle: (AxisData[VisuAxisNo].Axis_Standstill) <> 0
    Button (135,245 90x20), "Drive Halt"
        OnMouseUp: execute { arAxisCtrl_gb [VisuAxisNo].Admin._OpMode.en:=(ModeAh); }
    Rectangle (215,245 10x10), colour toggle: arAxisStatus_gb[VisuAxisNo].Admin._OpModeAck = ModeAH
    Button (135,275 90x20), "Disable"
        OnMouseUp: execute { arAxisCtrl_gb [VisuAxisNo].Admin._OpMode.en:=(ModeAb); }
    Rectangle (215,275 10x10), colour toggle: arAxisStatus_gb[VisuAxisNo].Admin._OpModeAck = ModeAB
    Rectangle (270,225 15x15), colour toggle: (AxisData[VisuAxisNo].Axis_InTorque) <> 0
    Rectangle (300,220 100x20), "In torque"
    Rectangle (270,305 135x15), text list: 'AxisMode', text index: arAxisStatus_gb [VisuAxisNo].Admin._OpModeAck
    Rectangle (415,300 150x20), "Actual operating mode"
    Rectangle (20,35 110x20), "Name of axis"
    Rectangle (345,35 70x20), "Drive Nr"
    Rectangle (115,35 215x20), "%s", text variable: arAxisStatus_gb [VisuAxisNo].Admin.Name
    Ellipse (80,65 20x20), colour toggle: arAxisStatus_gb [VisuAxisNo].Diag.Warning
    Rectangle (20,65 70x20), "Warning"
    Ellipse (155,65 20x20), colour toggle: arAxisStatus_gb [VisuAxisNo].Diag.Error
    Rectangle (105,65 40x20), "Error"
    Rectangle (180,65 60x20), "Error ID"
    Rectangle (250,65 220x20), text list: 'ErrorIDCode', text index: arAxisStatus_gb [VisuAxisNo].Diag.ErrorID
    Button (130,340 115x25), "Axis Overview"
        OnMouseUp:  Assign=Axis_Overview, Assign=Axis_Overview, Type=Assignment
    Button (260,340 115x25), "System Overview"
        OnMouseUp:  Assign=System_Overview_All_Axis, Assign=System_Overview_All_Axis, Type=Assignment
    Rectangle (425,35 80x20), "AXIS_%d", text variable: VisuAxisNo
        OnMouseUp: write VisuAxisNo via 
    Button (482,65 85x20), "Clear error"
        tap arAxisCtrl_gb [VisuAxisNo].Admin.ClearError
    Rectangle (557,65 10x10), colour toggle: arAxisCtrl_gb [VisuAxisNo].Admin.ClearError
END_VISUALIZATION

// IndraMotionMlc1/Application/AxisInterface/Visualizations/AxisModes/Velocity_mode
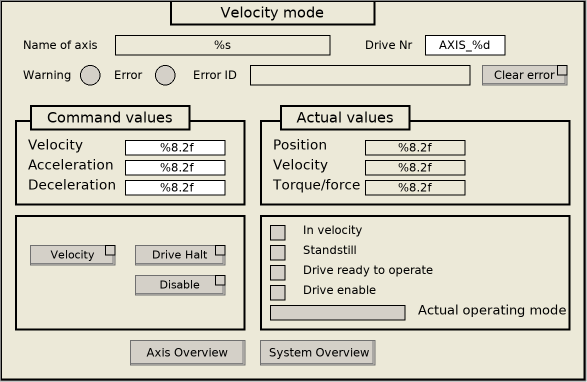
VISUALIZATION Velocity_mode  // 587x382
    Rectangle (0,0 585x380)
    Rectangle (15,215 230x115)
    Rectangle (15,120 230x85)
    Rectangle (30,105 160x25), "Command values"
    Rectangle (25,135 80x20), "Velocity"
    Rectangle (25,155 100x20), "Acceleration"
    Rectangle (25,175 100x20), "Deceleration"
    Rectangle (125,160 100x15), "%8.2f", text variable: arAxisCtrl_gb [VisuAxisNo].VelMode.Acceleration
        OnMouseUp: write arAxisCtrl_gb [VisuAxisNo].VelMode.Acceleration via 
    Rectangle (125,180 100x15), "%8.2f", text variable: arAxisCtrl_gb [VisuAxisNo].VelMode.Deceleration
        OnMouseUp: write arAxisCtrl_gb [VisuAxisNo].VelMode.Deceleration via 
    Rectangle (125,140 100x15), "%8.2f", text variable: arAxisCtrl_gb [VisuAxisNo].VelMode.Velocity
        OnMouseUp: write arAxisCtrl_gb [VisuAxisNo].VelMode.Velocity via Edit
    Rectangle (260,120 310x85)
    Rectangle (280,105 130x25), "Actual values"
    Rectangle (270,135 70x20), "Position"
    Rectangle (270,155 75x20), "Velocity"
    Rectangle (270,175 90x20), "Torque/force"
    Rectangle (365,160 100x15), "%8.2f", text variable: AxisData[VisuAxisNo].rActualVelocity_i
    Rectangle (365,180 100x15), "%8.2f", text variable: AxisData[VisuAxisNo].rActualTorqueForce_i
    Rectangle (365,140 100x15), "%8.2f", text variable: AxisData[VisuAxisNo].rActualPosition_i
    Rectangle (170,0 205x25), "Velocity mode"
    Button (30,245 85x20), "Velocity"
        OnMouseUp: execute { arAxisCtrl_gb[VisuAxisNo].Admin._OpMode.en:=(ModeVel); }
    Rectangle (105,245 10x10), colour toggle: (arAxisStatus_gb[VisuAxisNo].Admin.MODE_VEL) <> 0
    Rectangle (260,215 310x115)
    Rectangle (300,240 100x20), "Standstill"
    Rectangle (270,285 15x15), colour toggle: (AxisData[VisuAxisNo].Axis_Power) <> 0
    Rectangle (270,265 15x15), colour toggle: (AxisData[VisuAxisNo].Axis_InAb) <> 0
    Rectangle (300,280 170x20), "Drive enable"
    Rectangle (300,260 190x20), "Drive ready to operate"
    Rectangle (270,245 15x15), colour toggle: (AxisData[VisuAxisNo].Axis_Standstill) <> 0
    Button (135,245 90x20), "Drive Halt"
        OnMouseUp: execute { arAxisCtrl_gb [VisuAxisNo].Admin._OpMode.en:=(ModeAh); }
    Rectangle (215,245 10x10), colour toggle: (arAxisStatus_gb[VisuAxisNo].Admin.MODE_AH) <> 0
    Button (135,275 90x20), "Disable"
        OnMouseUp: execute { arAxisCtrl_gb [VisuAxisNo].Admin._OpMode.en:=(ModeAb); }
    Rectangle (215,275 10x10), colour toggle: (arAxisStatus_gb[VisuAxisNo].Admin._OpModeAck = ModeAb) <> 0
    Rectangle (270,225 15x15), colour toggle: (AxisData[VisuAxisNo].Axis_InVelocity) <> 0
    Rectangle (300,220 100x20), "In velocity"
    Rectangle (270,305 135x15), text list: 'AxisMode', text index: arAxisStatus_gb [VisuAxisNo].Admin._OpModeAck
    Rectangle (415,300 150x20), "Actual operating mode"
    Rectangle (20,35 110x20), "Name of axis"
    Rectangle (345,35 70x20), "Drive Nr"
    Rectangle (115,35 215x20), "%s", text variable: arAxisStatus_gb [VisuAxisNo].Admin.Name
    Ellipse (80,65 20x20), colour toggle: arAxisStatus_gb [VisuAxisNo].Diag.Warning
    Rectangle (20,65 70x20), "Warning"
    Ellipse (155,65 20x20), colour toggle: arAxisStatus_gb [VisuAxisNo].Diag.Error
    Rectangle (105,65 40x20), "Error"
    Rectangle (180,65 60x20), "Error ID"
    Rectangle (250,65 220x20), text list: 'ErrorIDCode', text index: arAxisStatus_gb [VisuAxisNo].Diag.ErrorID
    Button (130,340 115x25), "Axis Overview"
        OnMouseUp:  Assign=Axis_Overview, Assign=Axis_Overview, Type=Assignment
    Button (260,340 115x25), "System Overview"
        OnMouseUp:  Assign=System_Overview_All_Axis, Assign=System_Overview_All_Axis, Type=Assignment
    Rectangle (425,35 80x20), "AXIS_%d", text variable: VisuAxisNo
        OnMouseUp: write VisuAxisNo via 
    Button (482,65 85x20), "Clear error"
        tap arAxisCtrl_gb [VisuAxisNo].Admin.ClearError
    Rectangle (557,65 10x10), colour toggle: arAxisCtrl_gb [VisuAxisNo].Admin.ClearError
END_VISUALIZATION

// IndraMotionMlc1/Application/AxisInterface/Visualizations/ImcInterface/ImcControl
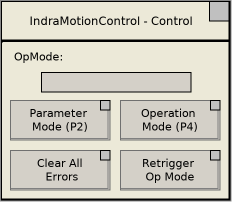
VISUALIZATION ImcControl  // 232x202
    Rectangle (0,0 230x200)
    Button (10,100 100x40), "Parameter Mode (P2)"
        OnMouseUp: execute { Global_ImcInterface.ImcCtrl .Admin._OpMode:=(IMC_MODE_CTRL_P2); }
    Rectangle (11,11 200x20), "IndraMotionControl - Control"
    Button (120,150 100x40), "Retrigger Op Mode"
        tap Global_ImcInterface.ImcCtrl .Admin.RetriggerOpMode
    Rectangle (210,150 10x10), colour toggle: Global_ImcInterface.ImcCtrl .Admin.RetriggerOpMode
    Rectangle (209,1 20x20), colour toggle: Global_ImcInterface.ImcStatus .InOperation
    Button (10,150 100x40), "Clear All Errors"
        tap Global_ImcInterface.ImcCtrl .Admin.ClearError
    Rectangle (100,150 10x10), colour toggle: Global_ImcInterface.ImcStatus .Diag.ClearErrorAck
    Rectangle (11,47 71x20), "OpMode:"
    Rectangle (41,72 150x20), text list: 'ImcModeControl', text index: Global_ImcInterface.ImcCtrl .Admin._OpMode
    Rectangle (100,100 10x10), colour toggle: (ImcCtrl.Admin._OpMode=IMC_MODE_CTRL_P2) <> 0
    Button (120,100 100x40), "Operation Mode (P4)"
        OnMouseUp: execute { Global_ImcInterface.ImcCtrl .Admin._OpMode:=(IMC_MODE_CTRL_BB); }
    Rectangle (210,100 10x10), colour toggle: (ImcCtrl.Admin._OpMode=IMC_MODE_CTRL_BB) <> 0
    Rectangle (1,40 229x1)
END_VISUALIZATION

// IndraMotionMlc1/Application/AxisInterface/Visualizations/ImcInterface/ImcInterface_Status_Control
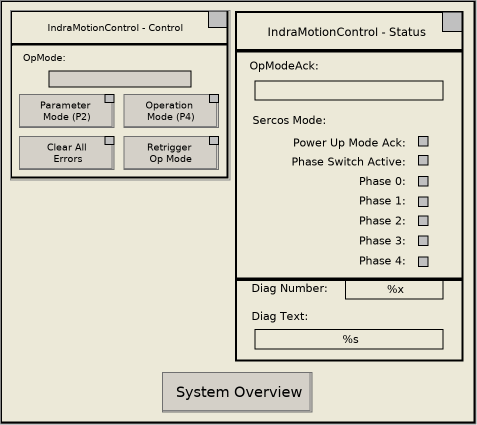
VISUALIZATION ImcInterface_Status_Control  // 477x425
    Rectangle (0,0 475x423)
    Button (162,372 150x40), "System Overview"
        OnMouseUp:  Assign=System_Overview_All_Axis, Assign=System_Overview_All_Axis, Type=Assignment
    Frame (10,10 220x170)
        shows ImcControl()
    Frame (235,11 230x352)
        shows ImcStatus()
END_VISUALIZATION

// IndraMotionMlc1/Application/AxisInterface/Visualizations/ImcInterface/ImcStatus
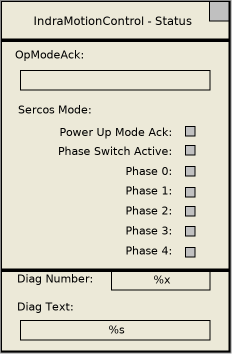
VISUALIZATION ImcStatus  // 232x354
    Rectangle (0,0 230x352)
    Rectangle (13,11 200x20), "IndraMotionControl - Status"
    Rectangle (209,1 20x20), colour toggle: Global_ImcInterface.ImcStatus .InOperation
    Rectangle (12,45 96x20), "OpModeAck:"
    Rectangle (20,70 190x20), text list: 'ImcModeStatus', text index: Global_ImcInterface.ImcStatus .Admin._OpModeAck
    Rectangle (0,40 230x0)
    Rectangle (15,100 90x20), "Sercos Mode:"
    Rectangle (0,270 230x0)
    Rectangle (185,187 10x10), colour toggle: Global_ImcInterface.ImcStatus .Admin.ModeStatus_P1
    Rectangle (185,226 10x10), colour toggle: Global_ImcInterface.ImcStatus .Admin.ModeStatus_P3
    Rectangle (185,206 10x10), colour toggle: Global_ImcInterface.ImcStatus .Admin.ModeStatus_P2
    Rectangle (185,166 10x10), colour toggle: Global_ImcInterface.ImcStatus .Admin.ModeStatus_P0
    Rectangle (185,247 10x10), colour toggle: Global_ImcInterface.ImcStatus .Admin.ModeStatus_BB
    Rectangle (185,145 10x10), colour toggle: Global_ImcInterface.ImcStatus .Admin.PhaseSwitchActive
    Rectangle (115,161 60x21), "Phase 0:"
    Rectangle (115,181 60x20), "Phase 1:"
    Rectangle (115,201 60x20), "Phase 2:"
    Rectangle (115,221 60x20), "Phase 3:"
    Rectangle (115,241 60x20), "Phase 4:"
    Rectangle (45,141 130x21), "Phase Switch Active:"
    Rectangle (45,125 130x15), "Power Up Mode Ack:"
    Rectangle (185,126 10x10), colour toggle: Global_ImcInterface.ImcStatus .Admin.PwrUpModeAck
    Rectangle (111,270 99x20), "%x", text variable: Global_ImcInterface.ImcStatus .Diag.Number
    Rectangle (20,320 190x20), "%s", text variable: Global_ImcInterface.ImcStatus .Diag.Message
    Rectangle (14,269 100x20), "Diag Number:"
    Rectangle (14,297 100x20), "Diag Text:"
END_VISUALIZATION

